// TwinCAT 3 PLC project Library
// Title: lcls-twincat-motion
// Company: SLAC
// ProjectVersion: 0.0.0
// ProgramVersion: 3.1.4026.17
// libraries:
//   LCLS General, * (SLAC)
//   lcls-twincat-math, * (SLAC - LCLS)
//   PMPS, * (SLAC - LCLS)
//   Tc2_EtherCAT, * (Beckhoff Automation GmbH)
//   Tc2_Math, * (Beckhoff Automation GmbH)
//   Tc2_MC2, * (Beckhoff Automation GmbH)
//   Tc2_Standard, * (Beckhoff Automation GmbH)
//   Tc2_System, * (Beckhoff Automation GmbH)
//   Tc2_Utilities, * (Beckhoff Automation GmbH)
//   Tc3_IPCDiag, * (Beckhoff Automation GmbH)
//   Tc3_JsonXml, * (Beckhoff Automation GmbH)
//   Tc3_Module, * (Beckhoff Automation GmbH)
//   TcUnit, * (www.tcunit.org)
// project tree:
//   DUTs/Deprecated/ ENUM_MotionRequest.TcDUT (not stored), DUT_MotionPneumaticActuator.TcDUT (not stored), DUT_MotionStage.TcDUT (not stored), DUT_PositionState.TcDUT (not stored), EL5042_Status.TcDUT (not stored), ENUM_EpicsHomeCmd.TcDUT (not stored), ENUM_EpicsInOut.TcDUT (not stored), ENUM_EpicsInOut_INT.TcDUT (not stored), ENUM_EpicsMotorCmd.TcDUT (not stored), ENUM_MotionFFType.TcDUT (not stored), ENUM_PnuematicActuatorPositionState.TcDUT (not stored), ENUM_StageBrakeMode.TcDUT (not stored), ENUM_StageEnableMode.TcDUT (not stored), ENUM_StatePMPSStatus.TcDUT (not stored)
//   DUTs/DS402/ ENUM_AxisStates.TcDUT (not stored), E_DS402DriveState.TcDUT, E_DS402EGU.TcDUT, E_DS402HomingMethod.TcDUT (not stored), E_DS402OpMode.TcDUT, E_HomeStates.TcDUT (not stored), E_Module.TcDUT (not stored), E_MoveMode.TcDUT (not stored), E_MoveState.TcDUT (not stored), ST_DS402Drive.TcDUT, ST_DS402DriveStatus.TcDUT
//   DUTs/ E_EpicsHomeCmd.TcDUT, ST_AxisParameterSetExposed.TcDUT (not stored), E_LCLSMotionError.TcDUT (not stored), E_MotionFFType.TcDUT (not stored), E_StatePMPSStatus.TcDUT (not stored), ST_MotionEpicsInterface.TcDUT, ST_MotionStage.TcDUT, ST_PositionState.TcDUT, ST_StateEpicsToPlc.TcDUT (not stored), ST_StatePlcToEpics.TcDUT (not stored), ST_StatePMPSEpicsToPlc.TcDUT (not stored), ST_EL5042_Status.TcDUT (not stored), E_EpicsInOut.TcDUT (not stored), E_EpicsMotorCmd.TcDUT, E_MotionRequest.TcDUT (not stored), E_StageBrakeMode.TcDUT (not stored), E_StageEnableMode.TcDUT (not stored), ST_MotionPneumaticActuator.TcDUT (not stored), E_PnuematicActuatorPositionState.TcDUT (not stored), ST_RenishawAbsEnc.TcDUT (not stored), ST_StatePMPSPlcToEpics.TcDUT (not stored)
//   GVLs/ MOTION_GVL.TcGVL (not stored), MotionConstants.TcGVL (not stored)
//   / PlcTask.TcTTO (not stored)
//   POUs/Deprecated/ FB_EpicsInOut.TcPOU (not stored), FB_PositionStateBase.TcPOU (not stored), FB_PositionStateBase_WithPMPS.TcPOU (not stored), FB_PositionStateBase_WithPMPS_Test.TcPOU (not stored), FB_PositionStateInOut.TcPOU (not stored), FB_PositionStateInOut_WithPMPS.TcPOU (not stored), FB_PositionStateInOut_WithPMPS_Test.TcPOU (not stored), FB_PositionStateManager.TcPOU (not stored), FB_PositionStatePMPS.TcPOU (not stored), FB_PositionStatePMPS_Base.TcPOU (not stored), FB_PositionStatePMPS_Test.TcPOU (not stored), FB_StatePTPMove.TcPOU (not stored)
//   POUs/ImplicitChecks/ CheckBounds.TcPOU (not stored), CheckDivDInt.TcPOU (not stored), CheckDivLInt.TcPOU (not stored), CheckDivLReal.TcPOU (not stored), CheckDivReal.TcPOU (not stored)
//   POUs/Motion/DS402/ FB_MotionStageE727.TcPOU, FB_MotionStageMCS2.TcPOU, I_DS402GenericDrive.TcIO
//   POUs/Motion/ FB_EncoderValue.TcPOU (not stored), FB_EncSaveRestore.TcPOU (not stored), FB_LogMotionError.TcPOU (not stored), FB_MotionBacklashCompensation.TcPOU (not stored), FB_MotionHoming.TcPOU (not stored), FB_MotionRequest.TcPOU (not stored), FB_MotionStage.TcPOU, FB_MotionStageNCParams.TcPOU (not stored), FB_MotionStageSim.TcPOU (not stored), FB_MotionPneumaticActuator.TcPOU (not stored), FB_MotionVirtualFrame.TcPOU (not stored)
//   POUs/Motion/Gantry/ FB_GantryAutoCoupling.TcPOU (not stored), FB_GantryDiffVirtualLimitSwitch.TcPOU (not stored)
//   POUs/Motion/PMPS/ FB_EncErrorFFO.TcPOU (not stored), FB_MiscStatesErrorFFO.TcPOU (not stored), FB_MotionBPTM.TcPOU (not stored), FB_MotionClearAsserts.TcPOU (not stored), FB_MotionReadPMPSDBND.TcPOU (not stored), FB_PerMotorFFOND.TcPOU (not stored), FB_NCErrorFFO.TcPOU (not stored), FB_PositionStatePMPS1D.TcPOU (not stored), FB_PositionStatePMPS2D.TcPOU (not stored), FB_PositionStatePMPS3D.TcPOU (not stored), FB_PositionStatePMPSND_Core.TcPOU (not stored), FB_Standard_PMPSDB.TcPOU (not stored), FB_StatePMPSEnables.TcPOU (not stored), FB_StatePMPSEnablesND.TcPOU (not stored)
//   POUs/Motion/States/Examples/ FB_PositionState1D_InOut.TcPOU (not stored), FB_PositionStatePMPS2D_InOut.TcPOU (not stored), FB_PositionStatePMPS1D_InOut.TcPOU (not stored), FB_PositionState2D_InOut.TcPOU (not stored)
//   POUs/Motion/States/ FB_PositionState2D.TcPOU (not stored), FB_PositionState3D.TcPOU (not stored), FB_PositionStateND_Core.TcPOU (not stored), FB_PositionStateMove.TcPOU (not stored), FB_PositionState1D.TcPOU (not stored), FB_PositionStateMoveND.TcPOU (not stored), FB_PositionStateRead.TcPOU (not stored), FB_PositionStateReadND.TcPOU (not stored), FB_StateSetupHelper.TcPOU (not stored), FB_StatesInputHandler.TcPOU (not stored)
//   POUs/Motion/States/Helpers/ FB_RawCountConverter.TcPOU (not stored), F_AtPositionState.TcPOU (not stored), F_PosOverLowerBound.TcPOU (not stored), F_PosUnderUpperBound.TcPOU (not stored), F_PosWithinDelta.TcPOU (not stored)
//   POUs/Motion/States/Internals/ FB_PositionStateInternal.TcPOU (not stored), FB_PositionStateInternalND.TcPOU (not stored), FB_PositionStateLock.TcPOU (not stored)
//   POUs/Motion/Utils/ FB_SetEnables.TcPOU (not stored), F_MotionErrorCodeLookup.TcPOU (not stored)
//   POUs/MotorTesting/ FB_MicroStepCountTest.TcPOU (not stored)
//   tc_mca_std_lib/DUTs/ DUT_AxisStatus_v0_01.TcDUT (not stored)
//   tc_mca_std_lib/GVLs/ GVL.TcGVL (not stored)
//   tc_mca_std_lib/POUs/ChangeConfig/ FB_ReadFloatParameter.TcPOU (not stored), FB_ReadParameterInNc_v1_00.TcPOU (not stored), FB_WriteFloatParameter.TcPOU (not stored), FB_WriteParameterInNc_v1_00.TcPOU (not stored)
//   tc_mca_std_lib/POUs/ErrorHandling/ DUT_ErrorState.TcDUT (not stored), DUT_TerminalError.TcDUT (not stored), FB_ErrorList.TcPOU (not stored), FB_TerminalError.TcPOU (not stored), GVL_ErrorSystem.TcGVL (not stored), ST_ErrorSystem.TcDUT (not stored)
//   tc_mca_std_lib/POUs/Hardware/EtherCAT_Terminals/Analog_Inputs/ EL3174_0002.TcPOU (not stored), EL3214.TcPOU (not stored), EL3255.TcPOU (not stored), FB_CalculateFrequency_3702_v0_01.TcPOU (not stored)
//   tc_mca_std_lib/POUs/Hardware/EtherCAT_Terminals/Digital_Inputs/ EL1008.TcPOU (not stored), EL1018.TcPOU (not stored), EL1808.TcPOU (not stored), EL1809.TcPOU (not stored), EL1819.TcPOU (not stored), FB_EL1252ASM_v1_00.TcPOU (not stored)
//   tc_mca_std_lib/POUs/Hardware/EtherCAT_Terminals/Digital_Outputs/ EL2014.TcPOU (not stored), EL2252.TcPOU (not stored), EL2808.TcPOU (not stored), EL2819.TcPOU (not stored)
//   tc_mca_std_lib/POUs/Hardware/EtherCAT_Terminals/Digital_Outputs/External_Types/ dutEL2521_Ctrl.TcDUT (not stored), dutEL2521_Status.TcDUT (not stored)
//   tc_mca_std_lib/POUs/Hardware/EtherCAT_Terminals/Measuring_Terminals/ EL5002.TcPOU (not stored), EL5021.TcPOU (not stored), EL5042.TcPOU (not stored), EL5101.TcPOU (not stored)
//   tc_mca_std_lib/POUs/Hardware/EtherCAT_Terminals/Motion/ EL7211_v1_00.TcPOU (not stored), EL9576_v1_00.TcPOU (not stored)
//   tc_mca_std_lib/POUs/Hardware/EtherCAT_Terminals/System/ EL9410.TcPOU (not stored), EL9505.TcPOU (not stored)
//   tc_mca_std_lib/POUs/Hardware/Other/ EK1200.TcPOU (not stored)
//   tc_mca_std_lib/POUs/Motion/ FB_DriveVirtual.TcPOU (not stored), FB_NcAxis.TcPOU (not stored)
//   tc_mca_std_lib/POUs/Motion/Homing/ FB_HomeDirect.TcPOU (not stored), FB_HomeFinish.TcPOU (not stored), FB_HomePrepare.TcPOU (not stored), FB_HomeReadNcVelocities.TcPOU (not stored), FB_HomeReadSoftLimEnable.TcPOU (not stored), FB_HomeToSwitch.TcPOU (not stored), FB_HomeVirtual.TcPOU (not stored), FB_HomeWriteNcVelocities.TcPOU (not stored), FB_HomeWriteSoftLimEnable.TcPOU (not stored)
//   Tests/ FB_AtPositionState_Test.TcPOU (not stored), FB_AxisParameterSetExposed_Test.TcPOU (not stored), FB_MiscStatesErrorFFO_Test.TcPOU (not stored), FB_MotionBPTM_Test.TcPOU (not stored), FB_MotionClearAsserts_Test.TcPOU (not stored), FB_MotionReadPMPSDBND_Test.TcPOU (not stored), FB_MotionVirtualFrame_Test.TcPOU (not stored), FB_NCErrorFFO_Test.TcPOU (not stored), FB_PerMotorFFOND_Test.TcPOU (not stored), FB_PositionStateMoveND_Test.TcPOU (not stored), FB_PositionStateMove_Test.TcPOU (not stored), FB_PositionStatePMPSND_Test.TcPOU (not stored), FB_PositionStateReadND_Test.TcPOU (not stored), FB_PositionStateRead_Test.TcPOU (not stored), FB_PositionStateND_Test.TcPOU (not stored), FB_PowerEnableMode_Test.TcPOU (not stored), FB_MotionBacklashCompensation_Test.TcPOU (not stored), FB_StatePMPSEnablesND_Test.TcPOU (not stored), FB_StatePMPSEnables_Test.TcPOU (not stored), FB_StateSetupHelper_Test.TcPOU (not stored), FB_TestHelperSetAndMove_Test.TcPOU (not stored), FB_TestStateInitTiming.TcPOU (not stored), PRG_TEST.TcPOU
//   Tests/Helpers/ E_TestStates.TcDUT (not stored), FB_CauseNCError.TcPOU (not stored), FB_MotionStageSetAndMoveHelper.TcPOU (not stored), FB_MotionStageSetHelper.TcPOU (not stored), FB_MotorTestSuite.TcPOU (not stored), FB_PMPSJsonTestHelper.TcPOU (not stored), FB_TestHelperSetAndMove.TcPOU (not stored)
// real-time tasks:
//   TASK PlcTask: cycle T#10ms, priority 20, ADS port 350
// motion (NC):
//   TASK NC-Task 1 SAF: cycle T#1ms, priority 4, ADS port 501
//   TASK NC-Task 1 SVB: cycle T#10ms, priority 8, ADS port 511
//   AXIS Axis_PositionStateRead_Test (id 3)
//   AXIS Axis_AtPositionState_Test (id 4)
//   AXIS Axis_TestHelperSetAndMove_Test (id 5)
//   AXIS Axis_PositionStateReadND_Test_1 (id 6)
//   AXIS Axis_PositionStateReadND_Test_2 (id 7)
//   AXIS Axis_PositionStateReadND_Test_3 (id 8)
//   AXIS Axis_PositionStateMove_Test (id 9)
//   AXIS Axis_PositionStateMoveND_Test_1 (id 10)
//   AXIS Axis_PositionStateMoveND_Test_2 (id 11)
//   AXIS Axis_PositionStateMoveND_Test_3 (id 12)
//   AXIS Axis_PositionStateND_Test_1 (id 13)
//   AXIS Axis_PositionStateND_Test_2 (id 14)
//   AXIS Axis_PositionStateND_Test_3 (id 15)
//   AXIS Axis_NCErrorFFO_Test (id 16)
//   AXIS Axis_PositionStatePMPSND_Test_1 (id 17)
//   AXIS Axis_PositionStatePMPSND_Test_2 (id 18)
//   AXIS Axis_PositionStatePMPSND_Test_3 (id 19)
//   AXIS Axis_StatePMPSEnable_Test (id 20)
//   AXIS Axis_PositionStateReadND_Test_4 (id 21)
//   AXIS Axis_PositionStateReadND_Test_5 (id 22)
//   AXIS Axis_TestStateInitTiming (id 1)
//   AXIS Axis_AxisParameter_Test (id 2)
//   AXIS Axis_PowerEnableMode_Test (id 29)
//   AXIS Axis_BacklashCompensation_Test (id 30)
//     OtherSettings: AllowMotionCmdToSlave=true
//     encoder EncType=1
//       ActPosCorrection: Enable=true
//     drive DrvType=5
//       Analog: TorqueSetpointScale=10, ScaleFactorActTorque=0.1
//       TimeComp: TaskDelayCycles=1
//     controller CtrType=1
//       CtrPara: PriorControlFactor=1
//         Observer: BandWidth=20
//   AXIS Axis_HomeNC_Test1 (id 32)
//     OtherSettings: AllowMotionCmdToSlave=true
//     encoder EncType=1
//     drive DrvType=5
//       Analog: TorqueSetpointScale=10, ScaleFactorActTorque=0.1
//       TimeComp: TaskDelayCycles=1
//     controller CtrType=1
//       CtrPara: PriorControlFactor=1
//         Observer: BandWidth=20
//   AXIS Axis_HomeNC_Test2 (id 33)
//     OtherSettings: AllowMotionCmdToSlave=true
//     encoder EncType=1
//     drive DrvType=5
//       Analog: TorqueSetpointScale=10, ScaleFactorActTorque=0.1
//       TimeComp: TaskDelayCycles=1
//     controller CtrType=1
//       CtrPara: PriorControlFactor=1
//         Observer: BandWidth=20
//   AXIS Axis_HomeNC_Test3 (id 34)
//     OtherSettings: AllowMotionCmdToSlave=true
//     encoder EncType=1
//     drive DrvType=5
//       Analog: TorqueSetpointScale=10, ScaleFactorActTorque=0.1
//       TimeComp: TaskDelayCycles=1
//     controller CtrType=1
//       CtrPara: PriorControlFactor=1
//         Observer: BandWidth=20
//   AXIS Axis_HomeNC_Test4 (id 35)
//     OtherSettings: AllowMotionCmdToSlave=true
//     encoder EncType=1
//     drive DrvType=5
//       Analog: TorqueSetpointScale=10, ScaleFactorActTorque=0.1
//       TimeComp: TaskDelayCycles=1
//     controller CtrType=1
//       CtrPara: PriorControlFactor=1
//         Observer: BandWidth=20
//   AXIS Axis_HomeNC_Test5 (id 36)
//     OtherSettings: AllowMotionCmdToSlave=true
//     encoder EncType=1
//     drive DrvType=5
//       Analog: TorqueSetpointScale=10, ScaleFactorActTorque=0.1
//       TimeComp: TaskDelayCycles=1
//     controller CtrType=1
//       CtrPara: PriorControlFactor=1
//         Observer: BandWidth=20
//   AXIS Axis_HomeNC_Test6 (id 37)
//     OtherSettings: AllowMotionCmdToSlave=true
//     encoder EncType=1
//     drive DrvType=5
//       Analog: TorqueSetpointScale=10, ScaleFactorActTorque=0.1
//       TimeComp: TaskDelayCycles=1
//     controller CtrType=1
//       CtrPara: PriorControlFactor=1
//         Observer: BandWidth=20
//   AXIS Axis_HomeNC_Test7 (id 38)
//     OtherSettings: AllowMotionCmdToSlave=true
//     encoder EncType=1
//     drive DrvType=5
//       Analog: TorqueSetpointScale=10, ScaleFactorActTorque=0.1
//       TimeComp: TaskDelayCycles=1
//     controller CtrType=1
//       CtrPara: PriorControlFactor=1
//         Observer: BandWidth=20
//   AXIS Axis_HomeNC_Test8 (id 39)
//     OtherSettings: AllowMotionCmdToSlave=true
//     encoder EncType=1
//     drive DrvType=5
//       Analog: TorqueSetpointScale=10, ScaleFactorActTorque=0.1
//       TimeComp: TaskDelayCycles=1
//     controller CtrType=1
//       CtrPara: PriorControlFactor=1
//         Observer: BandWidth=20
//   AXIS Axis_McMotionBlocks_Test1 (id 40)
//     OtherSettings: AllowMotionCmdToSlave=true
//     encoder EncType=1
//     drive DrvType=5
//       Analog: TorqueSetpointScale=10, ScaleFactorActTorque=0.1
//       TimeComp: TaskDelayCycles=1
//     controller CtrType=1
//       CtrPara: PriorControlFactor=1
//         Observer: BandWidth=20
//   AXIS Axis_McMotionBlocks_Test2 (id 41)
//     OtherSettings: AllowMotionCmdToSlave=true
//     encoder EncType=1
//     drive DrvType=5
//       Analog: TorqueSetpointScale=10, ScaleFactorActTorque=0.1
//       TimeComp: TaskDelayCycles=1
//     controller CtrType=1
//       CtrPara: PriorControlFactor=1
//         Observer: BandWidth=20
//   AXIS Axis_McMotionBlocks_Test3 (id 42)
//     OtherSettings: AllowMotionCmdToSlave=true
//     encoder EncType=1
//     drive DrvType=5
//       Analog: TorqueSetpointScale=10, ScaleFactorActTorque=0.1
//       TimeComp: TaskDelayCycles=1
//     controller CtrType=1
//       CtrPara: PriorControlFactor=1
//         Observer: BandWidth=20
//   AXIS Axis_McMotionBlocks_Test4 (id 43)
//     OtherSettings: AllowMotionCmdToSlave=true
//     encoder EncType=1
//     drive DrvType=5
//       Analog: TorqueSetpointScale=10, ScaleFactorActTorque=0.1
//       TimeComp: TaskDelayCycles=1
//     controller CtrType=1
//       CtrPara: PriorControlFactor=1
//         Observer: BandWidth=20
//   AXIS Axis_McMotionBlocks_Test5 (id 44)
//     OtherSettings: AllowMotionCmdToSlave=true
//     encoder EncType=1
//     drive DrvType=5
//       Analog: TorqueSetpointScale=10, ScaleFactorActTorque=0.1
//       TimeComp: TaskDelayCycles=1
//     controller CtrType=1
//       CtrPara: PriorControlFactor=1
//         Observer: BandWidth=20
//   AXIS Axis_McMotionBlocks_Test6 (id 45)
//     OtherSettings: AllowMotionCmdToSlave=true
//     encoder EncType=1
//       ActPosCorrection: Enable=true
//     drive DrvType=5
//       Analog: TorqueSetpointScale=10, ScaleFactorActTorque=0.1
//       TimeComp: TaskDelayCycles=1
//     controller CtrType=1
//       CtrPara: PriorControlFactor=1
//         Observer: BandWidth=20
//   AXIS Axis_McMotionBlocks_Test7 (id 46)
//     OtherSettings: AllowMotionCmdToSlave=true
//     encoder EncType=1
//       ActPosCorrection: Enable=true
//     drive DrvType=5
//       Analog: TorqueSetpointScale=10, ScaleFactorActTorque=0.1
//       TimeComp: TaskDelayCycles=1
//     controller CtrType=1
//       CtrPara: PriorControlFactor=1
//         Observer: BandWidth=20
//   AXIS Axis_McMotionBlocks_Test8 (id 47)
//     OtherSettings: AllowMotionCmdToSlave=true
//     encoder EncType=1
//       ActPosCorrection: Enable=true
//     drive DrvType=5
//       Analog: TorqueSetpointScale=10, ScaleFactorActTorque=0.1
//       TimeComp: TaskDelayCycles=1
//     controller CtrType=1
//       CtrPara: PriorControlFactor=1
//         Observer: BandWidth=20
//   AXIS Axis_MotionVirtualFrameRx_Test (id 23)
//   AXIS Axis_MotionVirtualFrameRy_Test (id 24)
//   AXIS Axis_MotionVirtualFrameRz_Test (id 25)
//   AXIS Axis_MotionVirtualFrameVx_Test (id 26)
//   AXIS Axis_MotionVirtualFrameVy_Test (id 27)
//   AXIS Axis_MotionVirtualFrameVz_Test (id 28)
// variable links:
//   Library Instance <-> NC-Task 1 SAF/Axes/Axis_AtPositionState_Test
//     PlcTask Inputs/PRG_TEST.fb_AtPositionState_Test.stMotionStage.Axis.NcToPlc <-> Outputs/ToPlc
//     PlcTask Outputs/PRG_TEST.fb_AtPositionState_Test.stMotionStage.Axis.PlcToNc <-> Inputs/FromPlc
//   Library Instance <-> NC-Task 1 SAF/Axes/Axis_AxisParameter_Test
//     PlcTask Inputs/PRG_TEST.fb_AxisParameterSetExposed_Test.stMotionStage.Axis.NcToPlc <-> Outputs/ToPlc
//     PlcTask Outputs/PRG_TEST.fb_AxisParameterSetExposed_Test.stMotionStage.Axis.PlcToNc <-> Inputs/FromPlc
//   Library Instance <-> NC-Task 1 SAF/Axes/Axis_BacklashCompensation_Test
//     PlcTask Inputs/PRG_TEST.fb_MotionBacklashCompensation_Test.stMotionStage.Axis.NcToPlc <-> Outputs/ToPlc
//     PlcTask Outputs/PRG_TEST.fb_MotionBacklashCompensation_Test.stMotionStage.Axis.PlcToNc <-> Inputs/FromPlc
//   Library Instance <-> NC-Task 1 SAF/Axes/Axis_MotionVirtualFrameRx_Test
//     PlcTask Inputs/PRG_TEST.fbMotionVirtualFrameTest.stMotionStageRx.Axis.NcToPlc <-> Outputs/ToPlc
//     PlcTask Outputs/PRG_TEST.fbMotionVirtualFrameTest.stMotionStageRx.Axis.PlcToNc <-> Inputs/FromPlc
//   Library Instance <-> NC-Task 1 SAF/Axes/Axis_MotionVirtualFrameRy_Test
//     PlcTask Inputs/PRG_TEST.fbMotionVirtualFrameTest.stMotionStageRy.Axis.NcToPlc <-> Outputs/ToPlc
//     PlcTask Outputs/PRG_TEST.fbMotionVirtualFrameTest.stMotionStageRy.Axis.PlcToNc <-> Inputs/FromPlc
//   Library Instance <-> NC-Task 1 SAF/Axes/Axis_MotionVirtualFrameRz_Test
//     PlcTask Inputs/PRG_TEST.fbMotionVirtualFrameTest.stMotionStageRz.Axis.NcToPlc <-> Outputs/ToPlc
//     PlcTask Outputs/PRG_TEST.fbMotionVirtualFrameTest.stMotionStageRz.Axis.PlcToNc <-> Inputs/FromPlc
//   Library Instance <-> NC-Task 1 SAF/Axes/Axis_MotionVirtualFrameVx_Test
//     PlcTask Inputs/PRG_TEST.fbMotionVirtualFrameTest.stMotionStageVx.Axis.NcToPlc <-> Outputs/ToPlc
//     PlcTask Outputs/PRG_TEST.fbMotionVirtualFrameTest.nPositionCountsVx <-> Enc/Inputs/In/nDataIn1
//     PlcTask Outputs/PRG_TEST.fbMotionVirtualFrameTest.stMotionStageVx.Axis.PlcToNc <-> Inputs/FromPlc
//   Library Instance <-> NC-Task 1 SAF/Axes/Axis_MotionVirtualFrameVy_Test
//     PlcTask Inputs/PRG_TEST.fbMotionVirtualFrameTest.stMotionStageVy.Axis.NcToPlc <-> Outputs/ToPlc
//     PlcTask Outputs/PRG_TEST.fbMotionVirtualFrameTest.nPositionCountsVy <-> Enc/Inputs/In/nDataIn1
//     PlcTask Outputs/PRG_TEST.fbMotionVirtualFrameTest.stMotionStageVy.Axis.PlcToNc <-> Inputs/FromPlc
//   Library Instance <-> NC-Task 1 SAF/Axes/Axis_MotionVirtualFrameVz_Test
//     PlcTask Inputs/PRG_TEST.fbMotionVirtualFrameTest.stMotionStageVz.Axis.NcToPlc <-> Outputs/ToPlc
//     PlcTask Outputs/PRG_TEST.fbMotionVirtualFrameTest.nPositionCountsVz <-> Enc/Inputs/In/nDataIn1
//     PlcTask Outputs/PRG_TEST.fbMotionVirtualFrameTest.stMotionStageVz.Axis.PlcToNc <-> Inputs/FromPlc
//   Library Instance <-> NC-Task 1 SAF/Axes/Axis_NCErrorFFO_Test
//     PlcTask Inputs/PRG_TEST.fb_NCErrorFFO_Test.stMotionStage.Axis.NcToPlc <-> Outputs/ToPlc
//     PlcTask Outputs/PRG_TEST.fb_NCErrorFFO_Test.stMotionStage.Axis.PlcToNc <-> Inputs/FromPlc
//   Library Instance <-> NC-Task 1 SAF/Axes/Axis_PositionStateMoveND_Test_1
//     PlcTask Inputs/PRG_TEST.fb_PositionStateMoveND_Test.astMotionStage[1].Axis.NcToPlc <-> Outputs/ToPlc
//     PlcTask Outputs/PRG_TEST.fb_PositionStateMoveND_Test.astMotionStage[1].Axis.PlcToNc <-> Inputs/FromPlc
//   Library Instance <-> NC-Task 1 SAF/Axes/Axis_PositionStateMoveND_Test_2
//     PlcTask Inputs/PRG_TEST.fb_PositionStateMoveND_Test.astMotionStage[2].Axis.NcToPlc <-> Outputs/ToPlc
//     PlcTask Outputs/PRG_TEST.fb_PositionStateMoveND_Test.astMotionStage[2].Axis.PlcToNc <-> Inputs/FromPlc
//   Library Instance <-> NC-Task 1 SAF/Axes/Axis_PositionStateMoveND_Test_3
//     PlcTask Inputs/PRG_TEST.fb_PositionStateMoveND_Test.astMotionStage[3].Axis.NcToPlc <-> Outputs/ToPlc
//     PlcTask Outputs/PRG_TEST.fb_PositionStateMoveND_Test.astMotionStage[3].Axis.PlcToNc <-> Inputs/FromPlc
//   Library Instance <-> NC-Task 1 SAF/Axes/Axis_PositionStateMove_Test
//     PlcTask Inputs/PRG_TEST.fb_PositionStateMove_Test.stMotionStage.Axis.NcToPlc <-> Outputs/ToPlc
//     PlcTask Outputs/PRG_TEST.fb_PositionStateMove_Test.stMotionStage.Axis.PlcToNc <-> Inputs/FromPlc
//   Library Instance <-> NC-Task 1 SAF/Axes/Axis_PositionStateND_Test_1
//     PlcTask Inputs/PRG_TEST.fb_PositionStateND_Test.stMotionStage1.Axis.NcToPlc <-> Outputs/ToPlc
//     PlcTask Outputs/PRG_TEST.fb_PositionStateND_Test.stMotionStage1.Axis.PlcToNc <-> Inputs/FromPlc
//   Library Instance <-> NC-Task 1 SAF/Axes/Axis_PositionStateND_Test_2
//     PlcTask Inputs/PRG_TEST.fb_PositionStateND_Test.stMotionStage2.Axis.NcToPlc <-> Outputs/ToPlc
//     PlcTask Outputs/PRG_TEST.fb_PositionStateND_Test.stMotionStage2.Axis.PlcToNc <-> Inputs/FromPlc
//   Library Instance <-> NC-Task 1 SAF/Axes/Axis_PositionStateND_Test_3
//     PlcTask Inputs/PRG_TEST.fb_PositionStateND_Test.stMotionStage3.Axis.NcToPlc <-> Outputs/ToPlc
//     PlcTask Outputs/PRG_TEST.fb_PositionStateND_Test.stMotionStage3.Axis.PlcToNc <-> Inputs/FromPlc
//   Library Instance <-> NC-Task 1 SAF/Axes/Axis_PositionStatePMPSND_Test_1
//     PlcTask Inputs/PRG_TEST.fb_PositionStatePMPSND_Test.stMotionStage1.Axis.NcToPlc <-> Outputs/ToPlc
//     PlcTask Outputs/PRG_TEST.fb_PositionStatePMPSND_Test.stMotionStage1.Axis.PlcToNc <-> Inputs/FromPlc
//   Library Instance <-> NC-Task 1 SAF/Axes/Axis_PositionStatePMPSND_Test_2
//     PlcTask Inputs/PRG_TEST.fb_PositionStatePMPSND_Test.stMotionStage2.Axis.NcToPlc <-> Outputs/ToPlc
//     PlcTask Outputs/PRG_TEST.fb_PositionStatePMPSND_Test.stMotionStage2.Axis.PlcToNc <-> Inputs/FromPlc
//   Library Instance <-> NC-Task 1 SAF/Axes/Axis_PositionStatePMPSND_Test_3
//     PlcTask Inputs/PRG_TEST.fb_PositionStatePMPSND_Test.stMotionStage3.Axis.NcToPlc <-> Outputs/ToPlc
//     PlcTask Outputs/PRG_TEST.fb_PositionStatePMPSND_Test.stMotionStage3.Axis.PlcToNc <-> Inputs/FromPlc
//   Library Instance <-> NC-Task 1 SAF/Axes/Axis_PositionStateReadND_Test_1
//     PlcTask Inputs/PRG_TEST.fb_PositionStateReadND_Test.astMotionStage[1].Axis.NcToPlc <-> Outputs/ToPlc
//     PlcTask Outputs/PRG_TEST.fb_PositionStateReadND_Test.astMotionStage[1].Axis.PlcToNc <-> Inputs/FromPlc
//   Library Instance <-> NC-Task 1 SAF/Axes/Axis_PositionStateReadND_Test_2
//     PlcTask Inputs/PRG_TEST.fb_PositionStateReadND_Test.astMotionStage[2].Axis.NcToPlc <-> Outputs/ToPlc
//     PlcTask Outputs/PRG_TEST.fb_PositionStateReadND_Test.astMotionStage[2].Axis.PlcToNc <-> Inputs/FromPlc
//   Library Instance <-> NC-Task 1 SAF/Axes/Axis_PositionStateReadND_Test_3
//     PlcTask Inputs/PRG_TEST.fb_PositionStateReadND_Test.astMotionStage[3].Axis.NcToPlc <-> Outputs/ToPlc
//     PlcTask Outputs/PRG_TEST.fb_PositionStateReadND_Test.astMotionStage[3].Axis.PlcToNc <-> Inputs/FromPlc
//   Library Instance <-> NC-Task 1 SAF/Axes/Axis_PositionStateReadND_Test_4
//     PlcTask Inputs/PRG_TEST.fb_PositionStateReadND_Test.astSqMotionStage[1].Axis.NcToPlc <-> Outputs/ToPlc
//     PlcTask Outputs/PRG_TEST.fb_PositionStateReadND_Test.astSqMotionStage[1].Axis.PlcToNc <-> Inputs/FromPlc
//   Library Instance <-> NC-Task 1 SAF/Axes/Axis_PositionStateReadND_Test_5
//     PlcTask Inputs/PRG_TEST.fb_PositionStateReadND_Test.astSqMotionStage[2].Axis.NcToPlc <-> Outputs/ToPlc
//     PlcTask Outputs/PRG_TEST.fb_PositionStateReadND_Test.astSqMotionStage[2].Axis.PlcToNc <-> Inputs/FromPlc
//   Library Instance <-> NC-Task 1 SAF/Axes/Axis_PositionStateRead_Test
//     PlcTask Inputs/PRG_TEST.fb_PositionStateRead_Test.stMotionStage.Axis.NcToPlc <-> Outputs/ToPlc
//     PlcTask Outputs/PRG_TEST.fb_PositionStateRead_Test.stMotionStage.Axis.PlcToNc <-> Inputs/FromPlc
//   Library Instance <-> NC-Task 1 SAF/Axes/Axis_PowerEnableMode_Test
//     PlcTask Inputs/PRG_TEST.fb_PowerEnableMode_Test.stMotionStage.Axis.NcToPlc <-> Outputs/ToPlc
//     PlcTask Outputs/PRG_TEST.fb_PowerEnableMode_Test.stMotionStage.Axis.PlcToNc <-> Inputs/FromPlc
//   Library Instance <-> NC-Task 1 SAF/Axes/Axis_StatePMPSEnable_Test
//     PlcTask Inputs/PRG_TEST.fb_StatePMPSEnables_Test.stMotionStage.Axis.NcToPlc <-> Outputs/ToPlc
//     PlcTask Outputs/PRG_TEST.fb_StatePMPSEnables_Test.stMotionStage.Axis.PlcToNc <-> Inputs/FromPlc
//   Library Instance <-> NC-Task 1 SAF/Axes/Axis_TestHelperSetAndMove_Test
//     PlcTask Inputs/PRG_TEST.fb_TestHelperSetAndMove_Test.stMotionStage.Axis.NcToPlc <-> Outputs/ToPlc
//     PlcTask Outputs/PRG_TEST.fb_TestHelperSetAndMove_Test.stMotionStage.Axis.PlcToNc <-> Inputs/FromPlc
//   Library Instance <-> NC-Task 1 SAF/Axes/Axis_TestStateInitTiming
//     PlcTask Inputs/PRG_TEST.fb_TestStateInitTiming.stMotionStage.Axis.NcToPlc <-> Outputs/ToPlc
//     PlcTask Outputs/PRG_TEST.fb_TestStateInitTiming.stMotionStage.Axis.PlcToNc <-> Inputs/FromPlc

// ---- DUTs/DS402/E_DS402DriveState.TcDUT
{attribute 'qualified_only'}
{attribute 'strict'}
{attribute 'to_string'}
TYPE E_DS402DriveState :
(
    INIT:=0,
    NO_FAULT:=1,
    SWITCH_ON_READY:=2,
    SWITCH_ON:=3,
    OPERATION_ENABLED:=4,
    FAULT:=5,
    FAULT_ACTIVE:=6,
    QUICK_STOP_ACTIVE:=7,
    SWITCH_ON_DISABLED:=8,
    MODE_ERROR:=9,
    WAIT	:= 10,
    DONE:=11
) UINT;
END_TYPE

// ---- DUTs/DS402/E_DS402EGU.TcDUT
{attribute 'qualified_only'}
{attribute 'strict'}
{attribute 'to_string'}
TYPE E_DS402EGU :
(
    MM:=0,
    UM:=1,
    NM:=2
);
END_TYPE

// ---- DUTs/DS402/E_DS402OpMode.TcDUT
{attribute 'qualified_only'}
{attribute 'strict'}
{attribute 'to_string'}
TYPE E_DS402OpMode :
(
    NONE:= 0,
    CALIBRATION:=-1,
    MCS2_OL_SM:=-4,
    PROFILE_POSITION:=1,
    HOMING:=6,
    CSP:=8
) SINT;
END_TYPE

// ---- DUTs/DS402/ST_DS402Drive.TcDUT
TYPE ST_DS402Drive:
STRUCT
    (* Global variables for the TPDO data from the drive. Each one is linked to the respective TPDO channel. *)
    stDS402DriveStatus 		AT %I*	: 	ST_DS402DriveStatus;
    nModeOfOperationDisplay AT %I*	: 	SINT;
    //nActualPosition 		AT %I*	: 	DINT;
    (*CSP drive mode*)
    nFollowingError 		AT %I*	: 	DINT;
    (* Global variables for the RPDO data to the drive. Each one is linked to the respective RPDO channel. *)
    // connected to I/O Task 'Control Word'
    nDS402DriveControl		AT %Q*	:	UINT;
    // Connected to NC task Ctrl 1 and Ctrl 2
    nDS402DriveControlNC	AT %I*	:	UINT;
    nTargetPosition 		AT %Q* 	: 	DINT;
    nModeOfOperation 		AT %Q* 	: 	SINT;
    nModeOfOperationNC 		AT %I* 	: 	SINT;
    (* Global variables for the RPDO data to the drive. Each one is linked to the respective RPDO channel. *)
    nProfilVelocity 		AT %Q* 	: 	DINT;
    nProfilAcceleration		AT %Q* 	: 	DINT;
    nProfilDecceleration	AT %Q* 	: 	DINT;
    nVelocityActualValue	AT %Q* 	: 	DINT;
    (* Global variables for the TPDO data from the drive. Each one is linked to the respective TPDO channel. *)
    nScantargetPosition		AT %Q*	: 	DINT;
    uScantargetVelocity		AT %Q*	: 	ULINT;
    (* Port Number of EtherCAT Slave *)
    nSlaveAddr	AT %I*  : UINT;
END_STRUCT
END_TYPE

// ---- DUTs/DS402/ST_DS402DriveStatus.TcDUT
TYPE ST_DS402DriveStatus :
    STRUCT
        ReadyToSwitchOn			: BIT; (* Bit 0 *)
        SwitchedOn				: BIT; (* Bit 1 *)
        OperationEnabled		: BIT; (* Bit 2 *)
        Fault					: BIT; (* Bit 3 *)
        VoltageEnabled			: BIT; (* Bit 4 *)
        QuickStopActive			: BIT; (* Bit 5 *)
        SwitchOnDisabled		: BIT; (* Bit 6 *)
        WarningCondition		: BIT; (* Bit 7 *)
        TrajectoryAborted		: BIT; (* Bit 8 *)
        RemoteCANopenControl	: BIT; (* Bit 9 *)
        TargetReached			: BIT; (* Bit 10 *)
        InternalLimitActive		: BIT; (* Bit 11 *)
        Bit12_OpModeSpecific	: BIT; (* Bit 12 *)
        Bit13_OpModeSpecific	: BIT; (* Bit 13 *)

    END_STRUCT
END_TYPE

// ---- DUTs/E_EpicsHomeCmd.TcDUT
{attribute 'qualified_only'}
{attribute 'strict'}
TYPE E_EpicsHomeCmd :
    // Defines the valid options for homing in FB_MotionStage
(
    LOW_LIMIT:=1, // Low limit switch
    HIGH_LIMIT:=2, // High limit switch
    HOME_VIA_LOW:=3, // Home switch via low switch
    HOME_VIA_HIGH:=4, // Home switch via high switch
    AUTO_ZERO	:= 5,	// Piezo Drives Homing
    ABSOLUTE_SET:=15, // Set here to be fHomePosition
    NONE:=-1 // Do not home, ever
);
END_TYPE

// ---- DUTs/ST_MotionEpicsInterface.TcDUT
TYPE ST_MotionEpicsInterface :
    // Defines the EPICS interface to moving a motor in TwinCAT
STRUCT
    // Name to use for log messages, fast faults, etc.
    sName: STRING;
    // Set to gantry difference tolerance
    nGantryTol: LINT:=0;
    // Encoder count at which this axis is aligned with other axis
    nEncRef: ULINT:=0;

    (* Commands *)
    // Used internally to request enables
    bEnable: BOOL;

    // Used internally to reset errors and other state
    {attribute 'pytmc' := '
        pv: PLC:bReset
        io: io
        field: ZNAM FALSE
        field: ONAM TRUE
        field: DESC Used internally to reset errors
    '}
    bReset: BOOL;
    // Used internally and by the IOC to start or stop a move
    bExecute: BOOL;

    (* Command Args *)
    // Used internally and by the IOC to pick what kind of move to do
    nCommand: INT;
    // Used internally and by the IOC to pass additional data to some commands
    nCmdData: INT;
    // Used internally and by the IOC to pick a destination for the move
    fPosition: LREAL;
    // Used internally and by the IOC to pick a move velocity
    fVelocity: LREAL;
    // Used internally and by the IOC to pick a move acceleration
    fAcceleration: LREAL;
    // Used internally and by the IOC to pick a move deceleration
    fDeceleration: LREAL;
    // Used internally and by the IOC to pick a home position
    {attribute 'pytmc' := '
        pv: PLC:fHomePosition
        io: io
        field: DESC Used internally and by the IOC to pick home position
    '}
    fHomePosition: LREAL;

    (* Info *)
    // Unique ID assigned to each axis in the NC
    nMotionAxisID: UDINT:=0;
    (* Returns *)
    // TRUE if in the middle of a command
    bBusy: BOOL;
    // TRUE if we've done a command and it has finished
    bDone: BOOL;
    // TRUE if the motor has been homed, or does not need to be homed
    bHomed: BOOL;

    // TRUE if we're in an error state
    {attribute 'pytmc' := '
        pv: PLC:bError
        io: i
        field: ZNAM FALSE
        field: ONAM TRUE
        field: DESC TRUE if we are in an error state
        update: 100Hz notify
    '}
    bError: BOOL;
    // Error code if nonzero
    {attribute 'pytmc' := '
        pv: PLC:nErrorId
        io: i
        field: DESC Error code if nonzero
        update: 100Hz notify
    '}
    nErrorId: UDINT;
    // Message to identify the error state
    {attribute 'pytmc' := '
        pv: PLC:sErrorMessage
        io: i
        field: DESC Message to identify the error state
        update: 100Hz notify
    '}
    sErrorMessage: STRING;

  // Misc axis status information for the IOC
    stAxisStatus: DUT_AxisStatus_v0_01;
END_STRUCT
END_TYPE

// ---- DUTs/ST_MotionStage.TcDUT
TYPE ST_MotionStage :
    // Defines the EPICS interface to moving a motor in TwinCAT
STRUCT
    (* Hardware *)

    // PLC Axis Reference
    Axis: AXIS_REF;
    // NC Forward Limit Switch: TRUE if ok to move
    bLimitForwardEnable AT %I*: BOOL;
    // NC Backward Limit Switch: TRUE if ok to move
    bLimitBackwardEnable AT %I*: BOOL;
    // NO Home Switch: TRUE if at home
    bHome AT %I*: BOOL;
    // NC Brake Output: TRUE to release brake
    bBrakeRelease AT %Q*: BOOL;
    // NC STO Input: TRUE if ok to move
    {attribute 'pytmc' := '
        pv: PLC:bHardwareEnable
        io: i
        field: ZNAM FALSE
        field: ONAM TRUE
        field: DESC TRUE if STO not hit
    '}
    bHardwareEnable AT %I*: BOOL;

    // Raw encoder IO for ULINT (Biss-C)
    nRawEncoderULINT AT %I*: ULINT;
    // Raw encoder IO for UINT (Relative Encoders)
    nRawEncoderUINT AT %I*: UINT;
    // Raw encoder IO for INT (LVDT)
    nRawEncoderINT AT %I*: INT;
    // Raw encoder IO for INT (EL5072 LVDT)
    nRawEncoderDINT AT %I*: DINT;

    (* Psuedo-hardware *)

    // Forward enable EPS summary
    bAllForwardEnable: BOOL:=FALSE;
    // Backward enable EPS summary
    bAllBackwardEnable: BOOL:=FALSE;
    // Enable EPS summary encapsulating emergency stop button and any additional motion preventive hardware
    bAllEnable: BOOL:=FALSE;
    // Forward virtual gantry limit switch
    bGantryForwardEnable: BOOL:=FALSE;
    // Backward virtual gantry limit switch
    bGantryBackwardEnable: BOOL:=FALSE;
    // Encoder count summary, if linked above
    {attribute 'pytmc' := '
        pv: PLC:nEncoderCount
        io: i
        field: DESC Count from encoder hardware
    '}
    nEncoderCount: UDINT;
    // Forward Enable EPS struct
    {attribute 'pytmc' := '
        pv: PLC:stEPSF
        io: i
        field: DESC Forward Enable Interlocks
    '}
    stEPSForwardEnable: DUT_EPS;
    // Backward Enable EPS struct
    {attribute 'pytmc' := '
        pv: PLC:stEPSB
        io: i
        field: DESC Backward Enable Interlocks
    '}
    stEPSBackwardEnable: DUT_EPS;
    // Power Enable EPS struct
    {attribute 'pytmc' := '
        pv: PLC:stEPSP
        io: i
        field: DESC Power Interlocks
    '}
    stEPSPowerEnable: DUT_EPS;

    (* Settings *)
    // Name to use for log messages, fast faults, etc.
    sName: STRING;
    // If TRUE, we want to enable the motor independently of PMPS or other safety systems.
    bPowerSelf: BOOL:=FALSE;
    // Determines when we automatically enable the motor
    nEnableMode: E_StageEnableMode:=E_StageEnableMode.DURING_MOTION;
    // Determines when we automatically disengage the brake
    nBrakeMode: E_StageBrakeMode:=E_StageBrakeMode.IF_ENABLED;
    // Determines our encoder homing strategy
    nHomingMode: E_EpicsHomeCmd:=E_EpicsHomeCmd.NONE;
    // Set true to activate gantry EPS
    bGantryAxis: BOOL:=FALSE;

    // Set to gantry difference tolerance
    nGantryTol: LINT:=0;

    // Encoder count at which this axis is aligned with other axis
    nEncRef: ULINT:=0;

    (* Commands *)
    // Used internally to request enables
    bEnable: BOOL;
    // Used internally to reset errors and other state
    {attribute 'pytmc' := '
        pv: PLC:bReset
        io: io
        field: ZNAM FALSE
        field: ONAM TRUE
        field: DESC Used internally to reset errors
    '}
    bReset: BOOL;
    // Used internally and by the IOC to start or stop a move
    bExecute: BOOL;
    // Used by the IOC to disable an axis
    {attribute 'pytmc' := '
        pv: PLC:bUserEnable
        io: io
        field: ZNAM DISABLE
        field: ONAM ENABLE
        field: DESC Used to disable power entirely for an axis
        autosave_pass1: VAL
    '}
    bUserEnable: BOOL := 1;

    (* Shortcut Commands *)
    // Start a move to fPosition with fVelocity
    bMoveCmd: BOOL;
    // Start the homing routine
    {attribute 'pytmc' := '
        pv: PLC:bHomeCmd
        io: io
        field: DESC Start the homing routine
    '}
    bHomeCmd: BOOL;

    (* Command Args *)
    // Used internally and by the IOC to pick what kind of move to do
    nCommand: INT;
    // Used internally and by the IOC to pass additional data to some commands
    nCmdData: INT;
    // Used internally and by the IOC to pick a destination for the move
    fPosition: LREAL;
    // Used internally and by the IOC to pick a move velocity
    fVelocity: LREAL;
    // Used internally and by the IOC to pick a move acceleration
    fAcceleration: LREAL;
    // Used internally and by the IOC to pick a move deceleration
    fDeceleration: LREAL;
    // Used internally and by the IOC to pick a home position
    {attribute 'pytmc' := '
        pv: PLC:fHomePosition
        io: io
        field: DESC Used internally and by the IOC to pick home position
        autosave_pass1: VAL
    '}
    fHomePosition: LREAL;

    (* Info *)
    // Unique ID assigned to each axis in the NC
    nMotionAxisID: UDINT:=0;

    (* Returns *)
    // TRUE if done enabling
    bEnableDone: BOOL;
    // TRUE if in the middle of a command
    bBusy: BOOL;
    // TRUE if we've done a command and it has finished
    bDone: BOOL;
    // TRUE if the motor has been homed, or does not need to be homed
    bHomed: BOOL;
    // TRUE if we have safety permission to move
    bSafetyReady: BOOL;
    // TRUE if we're in an error state
    {attribute 'pytmc' := '
        pv: PLC:bError
        io: i
        field: ZNAM FALSE
        field: ONAM TRUE
        field: DESC TRUE if we are in an error state
    '}
    bError: BOOL;
    // Error code if nonzero
    {attribute 'pytmc' := '
        pv: PLC:nErrorId
        io: i
        field: DESC Error code if nonzero
    '}
    nErrorId: UDINT;
    // Message to identify the error state
    {attribute 'pytmc' := '
        pv: PLC:sErrorMessage
        io: i
        field: DESC Message to identify the error state
    '}
    sErrorMessage: STRING;
    // Internal hook for custom error messages
    sCustomErrorMessage: STRING;
    // MC_ReadParameterSet Output
    stAxisParameters: ST_AxisParameterSet;
    // NC parameters that are exposed with pytmc pragmas
    {attribute 'pytmc' := '
        pv: PLC:AxisPar
        io: i
        field: DESC Axis configuration parameters in the numerical controller.
    '}
    stAxisParametersExposed: ST_AxisParameterSetExposed;
    // True if we've updated stAxisParameters at least once
    bAxisParamsInit: BOOL;

    // Misc axis status information for the IOC
    stAxisStatus: DUT_AxisStatus_v0_01;

    (* Other status information for users of the IOC *)
    // Position lag difference
    {attribute 'pytmc' := '
        pv: PLC:fPosDiff
        io: i
        field: DESC Position lag difference
    '}
    fPosDiff: LREAL;

    (* Backlash compensation*)
    // Enabled axis backlash compensation
    {attribute 'pytmc' := '
        pv: PLC:bBacklashEn
        io: io
        field: ZNAM FALSE
        field: ONAM TRUE
        field: DESC Enable Backlash compensation
        autosave_pass1: VAL
    '}
    bUserBacklashEn: BOOL;

    // backlash compensation status
    {attribute 'pytmc' := '
        pv: PLC:bBacklasStatus
        io: i
        field: ZNAM DISABLED
        field: ONAM ENABLED
        field: DESC Backlash compensation status
    '}
    bBacklashStatus: BOOL;

    // Backlash compensation value
    {attribute 'pytmc' := '
        pv: PLC:fBacklash
        io: io
        field: DESC Backlash compensation
        autosave_pass1: VAL
    '}
    fBacklash: LREAL;

    // Current Backlash compensation value ?
    {attribute 'pytmc' := '
        pv: PLC:fCurrentBacklash
        io: i
        field: DESC Currently applied compensation
    '}
    fCurrentBacklash: LREAL;
END_STRUCT
END_TYPE

// ---- DUTs/ST_PositionState.TcDUT
TYPE ST_PositionState :
    // Defines settings and current safety status for moves to specific positions for an axis
STRUCT
    // Name as queried via the NAME PV in EPICS
    {attribute 'pytmc' := '
        pv: NAME
        io: input
        field: DESC Name of this position state
    '}
    sName: STRING := 'Invalid';

    // Position associated with this state
    {attribute 'pytmc' := '
        pv: SETPOINT
        io: io
        field: DESC Axis position associated with this state
        autosave_pass1: VAL
    '}
    fPosition: LREAL;

    {attribute 'pytmc' := '
        pv: ENCODER
        io: i
        field: DESC Encoder count associated with this state
    '}
    nEncoderCount: UDINT;

    // Maximum allowable deviation from fPosition while at the state
    fDelta: LREAL;

    // Speed at which to move to this state
    {attribute 'pytmc' := '
        pv: VELO
        io: io
        field: DESC Speed at which to move to this state
        autosave_pass1: VAL
    '}
    fVelocity: LREAL;

    // (optional) Acceleration to use for moves to this state
    fAccel: LREAL;

    // (optional) Deceleration to use for moves to this state
    fDecel: LREAL;

    // Safety parameter. This must be set to TRUE by the PLC program to allow moves to this state. This is expected to change as conditions change.
    {attribute 'pytmc' := '
        pv: MOVE_OK
        io: i
        field: ZNAM FALSE
        field: ONAM TRUE
        field: DESC TRUE if the move would be safe
    '}
    bMoveOk: BOOL;

    // Signifies to FB_PositionStateLock that this state should be immutable
    bLocked: BOOL;

    // Set this to TRUE when you make your state. This defaults to FALSE so that uninitialized states can never be moved to
    bValid: BOOL;

    // Set this to TRUE when you want to use the raw encoder counts to define the state
    bUseRawCounts: BOOL;

    // Is set to TRUE by FB_PositionStateInternal when called
    bUpdated: BOOL;

    // We give this a state name and it is used to load parameters from the pmps database.
    stPMPS: ST_DbStateParams;
END_STRUCT
END_TYPE

// ---- DUTs/E_EpicsMotorCmd.TcDUT
{attribute 'qualified_only'}
{attribute 'strict'}
TYPE E_EpicsMotorCmd :
    // Defines valid EPICS commands for nCommand
(
    JOG := 0,
    MOVE_VELOCITY := 1,
    MOVE_RELATIVE := 2,
    MOVE_ABSOLUTE := 3,
    MOVE_MODULO := 4,
    HOME := 10,
    GEAR := 30,
	CALIBRATE:=40
);
END_TYPE

// ---- POUs/Motion/DS402/I_DS402GenericDrive.TcIO
INTERFACE I_DS402GenericDrive

METHOD ExposedParameters
VAR_INPUT
	Enable : BOOL; 
    tRefreshDelay: TIME;
END_VAR
END_METHOD

METHOD Home
VAR_INPUT
    Enable 				: BOOL;
END_VAR
END_METHOD

METHOD ModeOperation
VAR_INPUT
END_VAR
END_METHOD

METHOD MoveAbsolute
VAR_INPUT
END_VAR
END_METHOD

METHOD PersistParameters
VAR_INPUT
	 Enable: BOOL;
END_VAR
END_METHOD

METHOD Power : BOOL
VAR_INPUT
END_VAR
END_METHOD

METHOD ReadDriveCodes : BOOL
END_METHOD

METHOD Reset : BOOL
VAR_INPUT
END_VAR
END_METHOD

METHOD RestoreMotionParams
VAR_INPUT
    Enable	: BOOL;
END_VAR
END_METHOD

METHOD ScaleDriveParams
VAR_INPUT
END_VAR
END_METHOD

METHOD ScaleEncRawValue
VAR_INPUT
END_VAR
END_METHOD

METHOD ScaleHomingParams
VAR_INPUT
END_VAR
END_METHOD

METHOD ScaleJogParams
VAR_INPUT
END_VAR
END_METHOD

METHOD SetChanParams
VAR_INPUT
    Enable : BOOL;
END_VAR
END_METHOD

METHOD SetEnables
VAR_INPUT
END_VAR
END_METHOD

METHOD SetEpicsStatus
VAR_INPUT
END_VAR
END_METHOD

METHOD SetJogParams
VAR_INPUT
	Enable : BOOL;
END_VAR
END_METHOD

METHOD StateMachine
VAR_INPUT
	Enable : BOOL;
END_VAR
END_METHOD

METHOD  StepMove
VAR_INPUT
	Enable : BOOL;
END_VAR
END_METHOD

METHOD WriteParameterNC
VAR_INPUT
    Execute:BOOL;
    ParameterNumber : MC_AxisParameter;
    ParameterValue	: LREAL;
END_VAR
END_METHOD

END_INTERFACE

// ---- POUs/Motion/DS402/FB_MotionStageE727.TcPOU
(*	MCS2 Motion Stage . Controller a stage in CSP (NC), STEP_MODE and Homing via DS402 interface
     Using an overriden Position Holding timer. power enable mode must be 'DURING_MOTION'. for close loop aka CSP control
    set bServo PV to true, fort open loop step mode bServo must be cleared
*)
{attribute 'call_after_init'}
FUNCTION_BLOCK FB_MotionStageE727 IMPLEMENTS I_DS402GenericDrive
VAR
    {attribute 'no_copy'}
    stMotionStage  : REFERENCE TO ST_MotionStage;
    // Hardware I/O
    stDS402Drive 		: ST_DS402Drive;
    // Must be Provided
    {attribute 'hide'}
    eModule 			: E_Module;
    {attribute 'hide'}
    eHomeMode			: E_EpicsHomeCmd :=E_EpicsHomeCmd.AUTOZERO;
    {attribute 'hide'}
    eBufferMode 		: MC_BufferMode := MC_BufferMode.MC_Aborting;
    {attribute 'hide'}
    eMotionState 		: E_MoveState;
    {attribute 'hide'}
    eHomeState  		: E_MoveState;
    {attribute 'hide'}
    fbMcPower 			: MC_Power;
    {attribute 'hide'}
    fbMcMoveAbsolute 	: MC_MoveAbsolute;
    {attribute 'hide'}
    fbMcHalt 			: MC_Halt;
    {attribute 'hide'}
    fbMcReset 			: MC_Reset;
    {attribute 'hide'}
    fbMcWriteParameter 	: MC_WriteParameter;
    {attribute 'hide'}
    fbMcReadParams		: MC_ReadParameterSet;
    {attribute 'hide'}
    bEnPosLag 			: BOOL;
    {attribute 'hide'}
    bWrongParameter 	: BOOL;
    {attribute 'hide'}
    bExecMove 			: BOOL;
    {attribute 'hide'}
    bExecHome 			: BOOL;
    {attribute 'hide'}
    bNewMoveReq 		: BOOL;
    {attribute 'hide'}
    bHomeBusy 			: BOOL;
    {attribute 'hide'}
    bPrepareDisable 	: BOOL;
    {attribute 'hide'}
    bStop  				: BOOL;
    {attribute 'hide'}
    bOperational  		: BOOL;
    {attribute 'hide'}
    bLimOverride  		: BOOL;
    // use this for motion time axis states
    {attribute 'hide'}
    bLocalExec			: BOOL;
    // Save abd restore encoder value
    {attribute 'hide'}
    bInit				: BOOL;
    {attribute 'hide'}
    bHomeDone 			: BOOL;
    {attribute 'hide'}
    bHomeModeEnabled	: BOOL;
    {attribute 'hide'}
    bCSPModeEnabled		: BOOL;
    {attribute 'hide'}
    bRestoreLoad		: BOOL;
    {attribute 'hide'}
    bExecParamsRead		: BOOL;
    {attribute 'hide'}
    bCommandMoveAbsolute : BOOL;
    {attribute 'hide'}
    bRecentEnPosLagStatus 	: BOOL;
    {attribute 'hide'}
    bHomeAborted : BOOL;
    {attribute 'hide'}
    bDS402ManualEnabled : BOOL;
    {attribute 'hide'}
    fMeasuredVelo		: LREAL;
    {attribute 'hide'}
    fMeasuredAcc		: LREAL;
    {attribute 'hide'}
    fScalingFactor		: LREAL:= 0.000001;
    {attribute 'hide'}
    fParameterValue : LREAL;
    {attribute 'hide'}
    fMeasuredPos 		: LREAL;
    {attribute 'hide'}
    nSoftLimMin     	: LINT;
    {attribute 'hide'}
    nSoftLimMax     	: LINT;
    {attribute 'hide'}
    tonSyncHoming 		: TON;
    {attribute 'hide'}
    tonSlowParamReadTimer: TON;
    {attribute 'hide'}
    NCParamsTimer 		: TON;
    {attribute 'hide'}
    tonRestoreRetry		: TON;
    {attribute 'hide'}
    rtAborted 			: R_TRIG;
    {attribute 'hide'}
    rtStopDone			: R_TRIG;
    {attribute 'hide'}
    rtExec 				: R_TRIG;
    {attribute 'hide'}
    rtMoveCmdShortcut 	: R_TRIG;
    {attribute 'hide'}
    rtHomeCmdShortcut 	: R_TRIG;
    {attribute 'hide'}
    rtEnableMode    	: R_TRIG;
    {attribute 'hide'}
    rtUserExec      	: R_TRIG;
    {attribute 'hide'}
    rtModeChange      	: R_TRIG;
    {attribute 'hide'}
    rtMoveDone    		: R_TRIG;
    {attribute 'hide'}
    {attribute 'hide'}
    rtNewMoveReq  		: R_TRIG;
    {attribute 'hide'}
    ftExec      		: F_TRIG;
    {attribute 'hide'}
    rtHomeDone 			: R_TRIG;
    {attribute 'hide'}
    rtCSPModeOk			: R_TRIG;
    {attribute 'hide'}
    rtHomeModeEnable	: R_TRIG;
    {attribute 'hide'}
    nSubIndex			: BYTE := 0;
    {attribute 'hide'}
    nChanSoftwareLimIdx : WORD;
    {attribute 'hide'}
    nChanErrorCodeIdx 	: WORD;
    {attribute 'hide'}
    nChanSoftLimitIdx 	: WORD;
    {attribute 'hide'}
    bLocalReset: BOOL;
    {attribute 'hide'}
    nCommandLocal: INT := 3;
    {attribute 'hide'}
    nCmdDataLocal: INT;

END_VAR

VAR CONSTANT
    {attribute 'hide'}
    nChanSoftLimitBase	: WORD := 16#607D;
    {attribute 'hide'}
    nErrorCodeBase  	: WORD := 16#603F;
    // this true for SmartAct MCS2 and E-727.
    {attribute 'hide'}
    nChanOfsBase		: WORD := 16#800;

END_VAR

VAR PERSISTENT
    bSaved	: BOOL;
    fSavedPosition	: LREAL;
END_VAR

IF NOT __ISVALIDREF(stMotionStage) THEN
    RETURN;
END_IF

(* Done once after init*)
IF bInit THEN
    stMotionStage.nMotionAxisID := stMotionStage.Axis.NcToPlc.AxisId;
    (* Clear drive error/wraning condition, in open loop mode
       this will trigger a correct startup for procedure *)
    stDS402Drive.nDS402DriveControl := 128;
    // fist cycle reading of NC paramters
    bExecParamsRead := TRUE;
    bInit := FALSE;
END_IF
(* Check for the plc shortcut commands
   Used for testing or to circumvent motor record issues*)
rtMoveCmdShortcut(CLK:=stMotionStage.bMoveCmd);
rtHomeCmdShortcut(CLK:=stMotionStage.bHomeCmd);

(* Execute on rising edge*)
IF rtMoveCmdShortcut.Q AND NOT stMotionStage.bExecute THEN
    stMotionStage.bExecute:=TRUE;
    stMotionStage.nCommand := E_EpicsMotorCmd.MOVE_ABSOLUTE;
    bEnPosLag := bRecentEnPosLagStatus;
    fParameterValue := BOOL_TO_LREAL(bRecentEnPosLagStatus);

ELSIF rtHomeCmdShortcut.Q AND NOT stMotionStage.bExecute THEN
    stMotionStage.bExecute:= NOT ( stMotionStage.nCmdData=E_EpicsHomeCmd.ABSOLUTE_SET )
                            OR NOT ( stMotionStage.nCmdData=E_EpicsHomeCmd.NONE);
    stMotionStage.nCommand:=E_EpicsMotorCmd.HOME;
    (* Automatically fill the correct nCmdData for homing*)
    stMotionStage.nCmdData:=stMotionStage.nHomingMode;
    (*	Positional lag is not evaluated by E727 during homing, but NC does evaluated
        the condition which will lead to error as the lag is significant during homing
        disable the NC lag check and reenable it after homing is done
    *)
    IF stMotionStage.stAxisParameters.bCtrlEnablePosDiffControl.0 THEN
        bRecentEnPosLagStatus := stMotionStage.stAxisParameters.bCtrlEnablePosDiffControl.0;
        bEnPosLag := TRUE;
        fParameterValue := 0;
    END_IF

END_IF

(* entry point for local and EPICS main execs *)
rtUserExec(CLK:=stMotionStage.bExecute);
(* if a Move/Home Goal is comfirmed and there is no persistant
   error conditions, then we have a valid move request.*)
bNewMoveReq S= NOT stMotionStage.bBusy AND rtUserExec.Q AND NOT stMotionStage.bError;
(* this Move request is valid till an error occurs or the currently move is done *)
bNewMoveReq R= NOT stMotionStage.bExecute OR stMotionStage.bError;
bPrepareDisable R= bNewMoveReq;
rtNewMoveReq(CLK:=bNewMoveReq);
(* Moves are automatically allowed if no safety hooks.
   Otherwise, some other code will set this.*)
stMotionStage.bSafetyReady S= stMotionStage.bPowerSelf;
(* Set the proper command for the request move;
   if bservo not set, manual step moves will be performed *)
IF rtUserExec.Q THEN
    // Transfer nCommand and nCmdData to local copies at rising edge of bExecute (avoid issues if nCommand or nCmdData are changed during a command)
    nCmdDataLocal:=stMotionStage.nCmdData;
    nCommandLocal:=stMotionStage.nCommand;
    (* attempting to move an axis without homing first? *)
    IF stMotionStage.nHomingMode <> E_EpicsHomeCmd.NONE AND NOT stMotionStage.bHomed THEN
        (* one can just set bHome here even though no homing was done?*)
        stMotionStage.sErrorMessage:='Axis homing mode set, but homing routine pending';
    END_IF
END_IF

(* Set the drive in the correct operating mode. based on requested move command!
    NB: bservo must set for close loop motion
*)
ModeOperation();

(* NB: This is the only tested mode of operation so far. also aligned
    piezo drive position holding feature
*)
rtEnableMode(CLK:=(stMotionStage.nEnableMode = E_StageEnableMode.DURING_MOTION));
(* Handle auto-enable timing *)
CASE stMotionStage.nEnableMode OF
    (* Not recommended, not tested *)
    E_StageEnableMode.ALWAYS:
        stMotionStage.bEnable:=TRUE;
    E_StageEnableMode.DURING_MOTION:
        IF rtEnableMode.Q THEN
            stMotionStage.bEnable := FALSE;
        END_IF
        IF rtNewMoveReq.Q THEN
            (*MC block are not compatible with open loop Motion
                thus we wathc for correct close loop modes to use NC features *)
            stMotionStage.bEnable S= stMotionStage.bSafetyReady;
            bStop:=FALSE;
        END_IF
END_CASE
(*	Interlock mainly react on internal limit conditions inthe ove direction.
    MCS2 drive will go into error state when an internal limit is hit *)
Interlock();

IF bCSPModeEnabled THEN
    (*CSP using TwinCAT NC*)
    bLocalExec:= NOT stMotionStage.bError AND stMotionStage.bExecute AND stMotionStage.bAllEnable AND stMotionStage.bEnableDone AND stMotionStage.bSafetyReady;
ELSIF bHomeModeEnabled THEN
    bLocalExec:= NOT stMotionStage.bError AND stMotionStage.bExecute AND stMotionStage.bAllEnable AND  bOperational AND  stMotionStage.bSafetyReady;
ELSE
    bLocalExec:= FALSE;
END_IF

bExecHome:=bLocalExec AND stMotionStage.nCommand = 10;
bExecMove:=bLocalExec AND NOT bExecHome;

(* When we start, set the busy/done appropriately
   NB: CLose loop control using NC *)
rtExec(CLK:=bLocalExec);
IF rtExec.Q THEN
    // Release previous interruption if any
    stDS402Drive.nDS402DriveControl.8 := FALSE;
    stMotionStage.bDone := FALSE;
END_IF

(* updated axis status
   Not needed in manual mode *)
IF NOT bDS402ManualEnabled THEN
    stMotionStage.Axis.ReadStatus();
END_IF

(* Get a definitive bEnabled reading
   NB: use only in close loop mode, NC feature needed*)
CASE stMotionStage.Axis.Status.MotionState OF
    (* We are not enabled if there is an issue*)
    MC_AXISSTATE_UNDEFINED, MC_AXISSTATE_DISABLED, MC_AXISSTATE_ERRORSTOP:
        stMotionStage.bEnableDone := FALSE;
    ELSE
        stMotionStage.bEnableDone := TRUE;
END_CASE
//
IF stMotionStage.bReset THEN
    stMotionStage.bExecute:=FALSE;
    stMotionStage.bError := FALSE;
    stMotionStage.nErrorId := 0;
    stMotionStage.sErrorMessage:='';
    stMotionStage.sCustomErrorMessage:='';
    (*Manual Drive reset*)
    IF bDS402ManualEnabled THEN
        stDS402Drive.nDS402DriveControl := 128;
    ELSE
        bLocalReset := TRUE;
    END_IF

    stMotionStage.bReset:=FALSE;
END_IF

// Halt is always a user stop during motion
bStop S= NOT bLocalExec AND ((bHomeBusy AND (nCommandLocal=10)) OR (fbMcMoveAbsolute.Busy AND (nCommandLocal=3)));

//auto handle position lag monitoring, disable during homing.
WriteParameterNC(	Execute:=bEnPosLag,
                    ParameterNumber:=MC_AxisParameter.AxisEnPositionLagMonitoring,
                    ParameterValue:=fParameterValue);

(* Requested commands processing *)
CASE nCommandLocal OF
    E_EpicsMotorCmd.MOVE_ABSOLUTE:
        (*NC CSP Move Handling*)
        (* Trigger MC_Reset for close loop operation aka CSP mode *)
        Reset();
        Power();
        Halt();
        (*Wait for drive to be in the correct mode after a request was validated *)
        bCommandMoveAbsolute := bExecMove AND fbMcPower.Status AND bCSPModeEnabled;
        MoveAbsolute();
        (*IN CSP mode the drive control word is update via the NC
          Manual step mode and Homing will override this *)
         stDS402Drive.nDS402DriveControl := stDS402Drive.nDS402DriveControlNC;
    E_EpicsMotorCmd.HOME:
        (*DS402 Manual Homing*)
       Home(Enable:=TRUE);
END_CASE

stMotionStage.bBusy := bHomeBusy OR fbMcMoveAbsolute.Busy;

(* Check done moving via user stop, limit hit, Target Position reached, or from homing.*)
rtMoveDone(CLK:=fbMcMoveAbsolute.Done);
rtHomeDone(CLK:=bHomeDone);
rtStopDone(CLK:=fbMcHalt.Done);
rtAborted(CLK:=bHomeAborted);
IF rtAborted.Q OR rtStopDone.Q OR rtMoveDone.Q OR rtHomeDone.Q THEN
    IF NOT stMotionStage.bDone THEN
        stMotionStage.bHomed := bHomeDone;
        stMotionStage.bExecute:=FALSE;
        bCommandMoveAbsolute := FALSE;
        stMotionStage.bDone := fbMcMoveAbsolute.Done OR bHomeDone;
        IF bDS402ManualEnabled THEN
            // No standstill in Manual Mode
            stMotionStage.bEnable:=FALSE;
            (*Restore Postional lag monitoring*)
            bEnPosLag := FALSE;
        END_IF
        (* Release the internal limit override*)
        bLimOverride := FALSE;
        bHomeAborted := FALSE;
    END_IF
END_IF

(* updated axis status
   Not needed in manual mode *)
IF NOT bDS402ManualEnabled THEN
    stMotionStage.Axis.ReadStatus();
END_IF

ftExec(CLK:=stMotionStage.bExecute);
(*Handle auto-disable timing*)
bPrepareDisable S= stMotionStage.nEnableMode = E_StageEnableMode.DURING_MOTION AND ftExec.Q;
(* Delay the disable until we reach standstill *)
IF bPrepareDisable AND stMotionStage.Axis.Status.StandStill THEN
    bPrepareDisable:=FALSE;
    stMotionStage.bEnable:=FALSE;
END_IF

(* update encoder value and calibrated position*)
ScaleEncRawValue();
(*Drive parameters*)
ExposedParameters(Enable:=TRUE, tRefreshDelay:=T#2S);
(*Sync NC setting to drive settings*)
UpdateDriveMonitoringParams(Enable:=stMotionStage.bAxisParamsInit AND NOT stMotionStage.bBusy);
(* Save and restore as long as not an absolute encoder*)
PersistParameters( Enable:=stMotionStage.nHomingMode <> E_EpicsHomeCmd.NONE);
(*Restore encoder value at initialization*)
RestoreMotionParams(Enable:=stMotionStage.nHomingMode <> E_EpicsHomeCmd.NONE);

(*EPICS Motor record Update*)
UpdateEpicsStatus();
(*
    Error from functions and Nc. The error will send to EPICS interface based on predifined
    priority: axis, power, backlash, absoluteMove, etc...
*)
IF fbMcPower.Error AND fbMcPower.Active THEN
    stMotionStage.bError:=fbMcPower.Error;
    stMotionStage.nErrorId:=fbMcPower.ErrorID;
ELSIF fbMcMoveAbsolute.Error THEN
    stMotionStage.bError:=fbMcMoveAbsolute.Error;
    stMotionStage.nErrorId:=fbMcMoveAbsolute.ErrorID;
ELSIF fbMcHalt.Error AND fbMcHalt.Active THEN
    stMotionStage.bError:=fbMcHalt.Error;
    stMotionStage.nErrorId:=fbMcHalt.ErrorID;
ELSIF fbMcReset.Error  THEN
    stMotionStage.bError:=fbMcReset.Error;
    stMotionStage.nErrorId:=fbMcReset.ErrorID;
ELSIF fbMcWriteParameter.Error THEN
    stMotionStage.bError:=fbMcWriteParameter.Error;
    stMotionStage.nErrorId:=fbMcWriteParameter.ErrorID;
ELSIF fbMcReadParams.Error AND NOT stMotionStage.bBusy THEN
    stMotionStage.bError:=fbMcReadParams.Error;
    stMotionStage.nErrorId:=fbMcReadParams.ErrorID;
ELSE
    IF stMotionStage.bBusy THEN
        stMotionStage.sErrorMessage := '';
        stMotionStage.sCustomErrorMessage := '';
    END_IF
END_IF;

(*Double function, prioritize NC error otherwise read drive channel error code*)
ReadDriveCodes();

IF stMotionStage.sCustomErrorMessage <> ''
    AND stMotionStage.sErrorMessage = '' THEN
    stMotionStage.sErrorMessage := stMotionStage.sCustomErrorMessage;
END_IF

(*Clear motion flag when error occurs*)
IF stMotionStage.bError  THEN
    stMotionStage.bBusy := FALSE;
    stMotionStage.bDone := FALSE;
    stMotionStage.bEnable := FALSE;
END_IF

(* We've got the rising edge clear this flags.*)
stMotionStage.bMoveCmd:=FALSE;
stMotionStage.bHomeCmd:=FALSE;

METHOD PUBLIC  ExposedParameters
VAR_INPUT
    Enable : BOOL;
    tRefreshDelay: TIME;
END_VAR
// Periodic update of NC parameters
NCParamsTimer( IN:=Enable AND NOT bExecParamsRead, PT:=tRefreshDelay);
bExecParamsRead S= NCParamsTimer.Q;
fbMcReadParams(
    Parameter:=stMotionStage.stAxisParameters,
    Axis:=stMotionStage.Axis,
    Execute:= bExecParamsRead );

// Copy axis parameters that we want to expose to the EPICS layer.
stMotionStage.stAxisParametersExposed.bCtrlEnablePosDiffControl     := stMotionStage.stAxisParameters.bCtrlEnablePosDiffControl;
stMotionStage.stAxisParametersExposed.bEncEnableSoftEndMaxControl   := stMotionStage.stAxisParameters.bEncEnableSoftEndMaxControl;
stMotionStage.stAxisParametersExposed.bEncEnableSoftEndMinControl   := stMotionStage.stAxisParameters.bEncEnableSoftEndMinControl;
stMotionStage.stAxisParametersExposed.fAccelerationMax              := stMotionStage.stAxisParameters.fAccelerationMax;
stMotionStage.stAxisParametersExposed.fCtrlPosDiffMax               := stMotionStage.stAxisParameters.fCtrlPosDiffMax;
stMotionStage.stAxisParametersExposed.fCtrlPosDiffMaxTime           := stMotionStage.stAxisParameters.fCtrlPosDiffMaxTime;
stMotionStage.stAxisParametersExposed.fDecelerationMax              := stMotionStage.stAxisParameters.fDecelerationMax;
stMotionStage.stAxisParametersExposed.fEncSoftEndMax                := stMotionStage.stAxisParameters.fEncSoftEndMax;
stMotionStage.stAxisParametersExposed.fEncSoftEndMin                := stMotionStage.stAxisParameters.fEncSoftEndMin;
stMotionStage.stAxisParametersExposed.fVeloMaximum                  := stMotionStage.stAxisParameters.fVeloMaximum;
stMotionStage.stAxisParametersExposed.fEncOffset               		:= stMotionStage.stAxisParameters.fEncOffset;
stMotionStage.stAxisParametersExposed.fEncScaleFactorInternal       := stMotionStage.stAxisParameters.fEncScaleFactorInternal;

bExecParamsRead R= fbMcReadParams.Done OR fbMcReadParams.Error;
stMotionStage.bAxisParamsInit S= fbMcReadParams.Done;
END_METHOD

//FB_Init is always available implicitly and it is used primarily for initialization.
//The return value is not evaluated. For a specific influence, you can also declare the
//methods explicitly and provide additional code there with the standard initialization
//code. You can evaluate the return value.
METHOD FB_Init: BOOL
VAR_INPUT
    bInitRetains: BOOL; // TRUE: the retain variables are initialized (reset warm / reset cold)
    bInCopyCode: BOOL;  // TRUE: the instance will be copied to the copy code afterward (online change)
    stPiezoStage		:	REFERENCE TO ST_MotionStage;
    (*Mandatory must be unique for each MCS2 axis *)
    eModule : E_Module;
END_VAR
THIS^.stMotionStage REF= stPiezoStage;
THIS^.eModule := eModule;
END_METHOD

METHOD Halt : BOOL
fbMcHalt(
    Axis := stMotionStage.Axis,
    Execute := bStop AND bCSPModeEnabled,
    Deceleration := stMotionStage.fDeceleration,
    BufferMode := eBufferMode,
);
END_METHOD

METHOD PUBLIC Home
VAR_INPUT
    Enable 				: BOOL;
END_VAR
VAR_INST
    {attribute 'hide'}
    bMove 				: BOOL;
END_VAR
CASE eHomeMode OF
    E_EpicsHomeCmd.AUTOZERO:
        bMove S=  bExecHome;
    E_EpicsHomeCmd.NONE:
        bMove := FALSE;
        bHomeBusy :=  bExecHome;
        bHomeDone := NOT  bExecHome;
    ELSE
        bMove := FALSE;
END_CASE

IF bMove THEN
    CASE eHomeState OF
        // Wait for a rising edge
        E_MoveState.IDLING:
            IF bHomeModeEnabled AND bExecHome THEN
                bHomeDone := FALSE;
                bHomeBusy := TRUE;
                stMotionStage.bDone := FALSE;
                stDS402Drive.nDS402DriveControl:=15;
                eHomeState :=  E_MoveState.INIT;
            END_IF
        E_MoveState.INIT:
                        stDS402Drive.nDS402DriveControl.4:=1;
                                        eHomeState := E_MoveState.STARTED;
        E_MoveState.STARTED :
            // this is a comfirmation that routine is ongoing
            IF NOT stDS402Drive.stDS402DriveStatus.TargetReached
                AND NOT stDS402Drive.stDS402DriveStatus.Bit13_OpModeSpecific THEN
                bHomeBusy:=TRUE;
                bHomeDone:=FALSE;

                eHomeState:=E_MoveState.IN_PROGRESS;
            END_IF

        E_MoveState.IN_PROGRESS :

        IF bStop THEN
         stDS402Drive.nDS402DriveControl.8 :=1;
          bHomeAborted := TRUE;
          eHomeState:=E_MoveState.INTERRUPTED;

        // Genral Motion error i.e Following error ?
        ELSIF stDS402Drive.stDS402DriveStatus.Bit13_OpModeSpecific
                OR stDS402Drive.stDS402DriveStatus.WarningCondition THEN
            stMotionStage.bError := TRUE;
            eHomeState:=E_MoveState.ERROR;

        // Reached
        ELSIF stDS402Drive.stDS402DriveStatus.TargetReached
            AND stDS402Drive.stDS402DriveStatus.Bit12_OpModeSpecific
            AND NOT stDS402Drive.stDS402DriveStatus.Bit13_OpModeSpecific THEN
           eHomeState:=E_MoveState.DONE;
        END_IF
        E_MoveState.INTERRUPTED:
            bHomeBusy:=FALSE;
            eHomeState:=E_MoveState.IDLING;
        E_MoveState.DONE:
            bHomeBusy:=FALSE;
            bHomeDone:=TRUE;
            stMotionStage.fPosition:=0.0;

            IF (stMotionStage.nEnableMode = E_StageEnableMode.DURING_MOTION ) THEN
                stDS402Drive.nDS402DriveControl.4:=FALSE;

            ELSE
                stDS402Drive.nDS402DriveControl:=6;
            END_IF
            eHomeState:=E_MoveState.IDLING;
        E_MoveState.ERROR:
            bHomeDone:=FALSE;
            bHomeBusy:= FALSE;
            IF bWrongParameter THEN
                stMotionStage.sCustomErrorMessage:='Invalid motion Parameters';
                bWrongParameter := FALSE;
                stMotionStage.bError := TRUE;
            END_IF
            IF NOT stMotionStage.bError THEN
                eHomeState:=E_MoveState.IDLING;
            END_IF
    END_CASE
END_IF
END_METHOD

METHOD PUBLIC Interlock

VAR_INST
    {attribute 'hide'}
    bPositiveDirection  : BOOL;
    {attribute 'hide'}
    bNegativeDirection  : BOOL;
    {attribute 'hide'}
    ftForwardEnabled  	: F_TRIG;

    {attribute 'hide'}
    ftBackwardEnabled 	: F_TRIG;
END_VAR
// Positive or Negative direction
bPositiveDirection:=stMotionStage.bBusy AND stMotionStage.fPosDiff > 0;
bNegativeDirection:=stMotionStage.bBusy AND stMotionStage.fPosDiff < 0;

// For SmartAct MCS2 these limit are range and enstop limits. however a single bit in the status is used
// bLimOverride  : act as an override after limit was hit to allow reverse movement
stMotionStage.bLimitForwardEnable :=  bLimOverride OR NOT( bPositiveDirection AND stDS402Drive.stDS402DriveStatus.InternalLimitActive );
stMotionStage.bLimitBackwardEnable := bLimOverride OR NOT( bNegativeDirection AND stDS402Drive.stDS402DriveStatus.InternalLimitActive );

// use falling trigger to avoid spaming  sErrorMessage
ftForwardEnabled(CLK:=stMotionStage.bLimitForwardEnable);
ftBackwardEnabled(CLK:=stMotionStage.bLimitBackwardEnable);

IF  NOT bHomeBusy AND ftForwardEnabled.Q THEN
    // Not an error, just a warning
    stMotionStage.sCustomErrorMessage:='Cannot move past positive limit.';
    bLimOverride := TRUE;
END_IF

IF NOT bHomeBusy AND ftBackwardEnabled.Q THEN
    // Not an error, just a warning
    stMotionStage.sCustomErrorMessage:='Cannot move past Negative limit.';
    bLimOverride := TRUE;
END_IF

IF NOT stMotionStage.bError AND stMotionStage.bExecute AND NOT stMotionStage.bUserEnable THEN
    stMotionStage.bError := TRUE;
    stMotionStage.nErrorId := 1;
    stMotionStage.sCustomErrorMessage := 'Move requested, but user enable is disabled!';
END_IF

// Update all enable booleans
SetEnables();
END_METHOD

(*Switch the drive mod eof Operation
  Servo On: Profil Positioning or HOME
  Servo Off : STEP mode
*)
METHOD ModeOperation

VAR_INST
    tonSwitching : TON;
    bManualTransition: BOOL;
END_VAR
rtCSPModeOk(CLK:=( stDS402Drive.nModeOfOperationDisplay=E_DS402OpMode.CSP));
rtHomeModeEnable(CLK:=( stDS402Drive.nModeOfOperationDisplay=E_DS402OpMode.HOME));
// transition to close loop mode
IF rtCSPModeOk.Q THEN
    bHomeModeEnabled := FALSE;
    bCSPModeEnabled := TRUE;
ELSIF rtHomeModeEnable.Q THEN
    bHomeModeEnabled := TRUE;
    bCSPModeEnabled := FALSE;
    stDS402Drive.nDS402DriveControl := 0;
END_IF

IF rtUserExec.Q AND stMotionStage.bHomeCmd THEN
    IF (stDS402Drive.nModeOfOperationDisplay<>E_DS402OpMode.HOME) THEN
        stDS402Drive.nModeOfOperation := E_DS402OpMode.HOME;
        stDS402Drive.nDS402DriveControl := 128;
        // clear previous operational from switching away from this mode.
        bOperational := FALSE;
        bCSPModeEnabled := FALSE;
        bManualTransition := TRUE;
    ELSE
        bHomeModeEnabled := TRUE;
    END_IF
ELSIF rtUserExec.Q THEN
    IF (stDS402Drive.nModeOfOperationDisplay<>E_DS402OpMode.CSP) THEN
        stDS402Drive.nModeOfOperation := E_DS402OpMode.CSP;
        stDS402Drive.nDS402DriveControl := 128;
        bHomeModeEnabled := FALSE;
        bManualTransition := FALSE;
    ELSE
        bCSPModeEnabled := TRUE;
    END_IF
END_IF

bDS402ManualEnabled :=bHomeModeEnabled;
(*Handle correct startup procedure for manual move*)
StateMachine(Enable:=1);
END_METHOD

METHOD PUBLIC  MoveAbsolute

fbMcMoveAbsolute(
    Axis := stMotionStage.Axis,
    Execute := bCommandMoveAbsolute,
    Position := stMotionStage.fPosition,
    Velocity := stMotionStage.fVelocity,
    Acceleration := stMotionStage.fAcceleration,
    Deceleration := stMotionStage.fDeceleration,
    BufferMode := eBufferMode,
);
END_METHOD

METHOD PersistParameters
VAR_INPUT
    Enable	: BOOL;
END_VAR

VAR_INST
    {attribute 'hide'}
    bEncError			: BOOL;

    {attribute 'hide'}
    bRestoreWaitRetry	: BOOL;
END_VAR
// Save Encoder position
// needs some pre-conditions to use persistent storage
IF Enable THEN
    // Check ST_MotionStage for an encoder error (range 0x44nn)
    bEncError:= stMotionStage.Axis.Status.Error AND  ( stMotionStage.Axis.Status.ErrorID  >= 16#4400  AND stMotionStage.Axis.Status.ErrorID <= 16#44FF );
    // Do not save if we're currently loading or if there is an encoder error
    IF NOT bRestoreLoad AND NOT bEncError AND NOT bRestoreWaitRetry THEN
        fSavedPosition := stMotionStage.Axis.NcToPlc.ActPos;
        // This persistent variable lets us check if anything was saved
        // It will be TRUE at startup if we have saved values
        bSaved := TRUE;
        (*
            use this with a timer of a change threshold on the fActPosition
            to trigger a save from this PLC program. otherwise this will be a spamming
            persistence, filling up the disk.
        *)
        //iPersistentDataStorage.TriggerWriteOfPersistentData := bSaveEnabled;
    END_IF
END_IF
END_METHOD

{attribute 'call_after_init'}
(*	eModule: Mandatory must be unique for each MCS2 axis
    clears startup errors or warnings. the process is completed at run time
    SDO update of Drive and open Loop parameter Indexes based on module number
*)
METHOD PostInit
VAR_INPUT
END_VAR
(* SDO update of Drive and open Loop parameter Indexes based on module number*)
nChanErrorCodeIdx	:= nErrorCodeBase		+ ((eModule-1) * nChanOfsBase);
nChanSoftLimitIdx	:= nChanSoftLimitBase 	+ ((eModule-1) * nChanOfsBase);
bInit := TRUE;
END_METHOD

METHOD Power : BOOL
fbMcPower(
    Axis := stMotionStage.Axis,
    Enable := stMotionStage.bAllEnable AND bCSPModeEnabled,
    Enable_Positive := stMotionStage.bAllForwardEnable,
    Enable_Negative := stMotionStage.bAllBackwardEnable,
    Override := 100.0,
    BufferMode := eBufferMode );
END_METHOD

(* Read Drive error codes after a motion or fault condition occured *)
METHOD ReadDriveCodes : BOOL
VAR_INST
    {attribute 'hide'}
    fbErrorRead			: FB_EcCoESdoRead;
    {attribute 'hide'}
    nPiezoErrorCode   	: UDINT;
    {attribute 'hide'}
    fbLogError  		: FB_LogMotionError;
    {attribute 'hide'}
    ftErrorReadDone  	: F_TRIG;
END_VAR
fbErrorRead( sNetId:= THIS^.stMotionStage.stAxisParameters.sAmsNetId,
             nSlaveAddr:=stDS402Drive.nSlaveAddr,
             nIndex:=nChanErrorCodeIdx,
             nSubIndex :=nSubIndex,
             pDstBuf:= ADR(nPiezoErrorCode),
             cbBufLen:=SIZEOF(nPiezoErrorCode),
             bExecute:= stMotionStage.bError );

ftErrorReadDone(CLK:=fbErrorRead.bBusy);
IF ftErrorReadDone.Q THEN
    IF 	NOT fbErrorRead.bError AND nPiezoErrorCode <> 0 THEN
        stMotionStage.nErrorId := nPiezoErrorCode;
    END_IF
    stMotionStage.sErrorMessage := F_MotionErrorCodeLookup(nErrorId:=stMotionStage.nErrorId);
    fbLogError( stMotionStage:=stMotionStage, bEnable:=stMotionStage.bError);
END_IF
END_METHOD

METHOD Reset : BOOL
fbMcReset(
    Axis := stMotionStage.Axis,
    Execute := bLocalReset AND bCSPModeEnabled
);

IF fbMcReset.Done OR fbMcReset.Error THEN
    bLocalReset := FALSE;
END_IF
END_METHOD

METHOD RestoreMotionParams
VAR_INPUT
    Enable	: BOOL;
END_VAR

VAR_INST
    {attribute 'hide'}
    fbSetPos			: MC_SetPosition;
    {attribute 'hide'}
    bLoad				: BOOL;
    {attribute 'hide'}
    bRestoreDone 		: BOOL;
    {attribute 'hide'}
    bRestoreInit		: BOOL;
    {attribute 'hide'}
    bRestoreWaitRetry	: BOOL;
    {attribute 'hide'}
    nMaxRetries			: UINT := 10;
    {attribute 'hide'}
    nCurrTries			: UINT := 0;
    {attribute 'hide'}
    nLatchError			: UDINT;
END_VAR
IF Enable THEN
    // Trigger a load if anything was saved at all
    IF NOT bRestoreInit THEN
        bRestoreInit := TRUE;
        bRestoreLoad S= bSaved;
        fbSetPos.Options.ClearPositionLag := TRUE;
    END_IF

    // Set our position if bRestoreLoad is true
    fbSetPos( Axis:=stMotionStage.Axis, Execute:=bRestoreLoad, Position:=fSavedPosition);

    // Only load once, at startup
    bRestoreLoad R= fbSetPos.Done OR fbSetPos.Error;

    IF fbSetPos.Error THEN
        // Keep the error latched, it can disappear if Execute is set to FALSE
        nLatchError := fbSetPos.ErrorID;
        nCurrTries := nCurrTries + 1;
        IF nCurrTries >= nMaxRetries THEN
        // Alert the user that something has gone wrong
        stMotionStage.bError := TRUE;
        stMotionStage.nErrorId := nLatchError;
        stMotionStage.sCustomErrorMessage := 'Error loading previously saved position.';
        ELSE
            // Reset the FB for the next retry
            fbSetPos( Axis:=stMotionStage.Axis, Execute:=bRestoreLoad, Position:=fSavedPosition);
            // Try again
            bRestoreWaitRetry := TRUE;
        END_IF
    ELSE
        IF NOT bRestoreDone THEN
            stMotionStage.fPosition := fSavedPosition;
        END_IF
        bRestoreDone := TRUE;
    END_IF

    tonRestoreRetry( IN := bRestoreWaitRetry, PT := T#100MS);
    bRestoreLoad S= tonRestoreRetry.Q;
    bRestoreWaitRetry R= tonRestoreRetry.Q;
END_IF
END_METHOD

METHOD ScaleDriveParams
nSoftLimMax := LREAL_TO_DINT((stMotionStage.stAxisParameters.fEncSoftEndMax / MAX(stMotionStage.stAxisParameters.fEncScaleFactorInternal, fScalingFactor)));
nSoftLimMin := LREAL_TO_DINT((stMotionStage.stAxisParameters.fEncSoftEndMin / MAX(stMotionStage.stAxisParameters.fEncScaleFactorInternal, fScalingFactor)));
END_METHOD

METHOD ScaleEncRawValue
VAR_INPUT
  //  bEnable: BOOL;
END_VAR
(* SmartACT: The encoder count from the Piezo drive is not a raw count from the embeded actuator device
   we get a calibrated nm value. thus the use of abs() since this value is signed.
   PI: to be discovered *)
IF stMotionStage.nRawEncoderDINT <> 0 THEN
    stMotionStage.nEncoderCount:=DINT_TO_UDINT(ABS(stMotionStage.nRawEncoderDINT));
ELSE
    stMotionStage.nEncoderCount:=0;
END_IF

// calibrated encoder readback
fMeasuredPos:=stMotionStage.Axis.NcToPlc.ActPos;
fMeasuredVelo :=stMotionStage.Axis.NcToPlc.ActVelo;
fMeasuredAcc := stMotionStage.Axis.NcToPlc.ActAcc;
stMotionStage.fPosDiff:=stMotionStage.Axis.NcToPlc.PosDiff;
END_METHOD

(*Scale Home Move parameters*)
METHOD ScaleHomingParams
END_METHOD

(*Scaled Open Loop Step mode motion parameters*)
METHOD ScaleJogParams
VAR_INPUT
END_VAR
END_METHOD

{warning 'Add method implementation '}
METHOD SetChanParams
VAR_INPUT
    Enable	: BOOL;
END_VAR
END_METHOD

METHOD SetEnables
VAR_INPUT
END_VAR
stMotionStage.bAllForwardEnable:=stMotionStage.bLimitForwardEnable AND (stMotionStage.bGantryForwardEnable OR NOT stMotionStage.bGantryAxis) AND stMotionStage.stEPSForwardEnable.bEPS_OK;
stMotionStage.bAllBackwardEnable:=stMotionStage.bLimitBackwardEnable AND (stMotionStage.bGantryBackwardEnable OR NOT stMotionStage.bGantryAxis) AND stMotionStage.stEPSBackwardEnable.bEPS_OK;

stMotionStage.bAllEnable:=stMotionStage.bEnable AND stMotionStage.bHardwareEnable AND stMotionStage.stEPSPowerEnable.bEPS_OK;
stMotionStage.bAllEnable R= NOT stMotionStage.bUserEnable;
END_METHOD

{warning 'Add method implementation '}
METHOD SetEpicsStatus
END_METHOD

{warning 'Add method implementation '}
METHOD SetJogParams
VAR_INPUT
    Enable	: BOOL;
END_VAR
END_METHOD

METHOD StateMachine
VAR_INPUT
    Enable : BOOL;
END_VAR

VAR_INST
    rtFault: R_TRIG;
    {attribute 'hide'}
    bFault				: BOOL;
END_VAR
rtFault(CLK:=bFault);
(*switch on disable*)
IF NOT stDS402Drive.stDS402DriveStatus.ReadyToSwitchOn
    AND NOT stDS402Drive.stDS402DriveStatus.SwitchedOn
    AND NOT stDS402Drive.stDS402DriveStatus.OperationEnabled
    AND NOT stDS402Drive.stDS402DriveStatus.Fault
    AND stDS402Drive.stDS402DriveStatus.VoltageEnabled
    AND NOT stDS402Drive.stDS402DriveStatus.QuickStopActive
    AND  stDS402Drive.stDS402DriveStatus.SwitchOnDisabled THEN
        bOperational := FALSE;
        IF bDS402ManualEnabled AND NOT bStop  THEN
            THIS^.stDS402Drive.nDS402DriveControl := 6;
        END_IF
(*Ready to switch*)
ELSIF stDS402Drive.stDS402DriveStatus.ReadyToSwitchOn
    AND NOT stDS402Drive.stDS402DriveStatus.SwitchedOn
    AND NOT stDS402Drive.stDS402DriveStatus.OperationEnabled
    AND NOT stDS402Drive.stDS402DriveStatus.Fault
    AND stDS402Drive.stDS402DriveStatus.VoltageEnabled
    AND stDS402Drive.stDS402DriveStatus.QuickStopActive
    AND NOT stDS402Drive.stDS402DriveStatus.SwitchOnDisabled THEN
        bFault := FALSE;
        bOperational := FALSE;
        IF bDS402ManualEnabled AND NOT bStop  THEN
            THIS^.stDS402Drive.nDS402DriveControl := 7;
        END_IF
(*Switch on*)
ELSIF stDS402Drive.stDS402DriveStatus.ReadyToSwitchOn
    AND  stDS402Drive.stDS402DriveStatus.SwitchedOn
    AND NOT stDS402Drive.stDS402DriveStatus.OperationEnabled
    AND NOT stDS402Drive.stDS402DriveStatus.Fault
    AND stDS402Drive.stDS402DriveStatus.VoltageEnabled
    AND stDS402Drive.stDS402DriveStatus.QuickStopActive
    AND NOT stDS402Drive.stDS402DriveStatus.SwitchOnDisabled THEN
        bOperational := FALSE;
        IF bDS402ManualEnabled AND NOT bStop  THEN
            THIS^.stDS402Drive.nDS402DriveControl := 15;
        END_IF
(*Operation enbaled*)
ELSIF stDS402Drive.stDS402DriveStatus.ReadyToSwitchOn
    AND stDS402Drive.stDS402DriveStatus.SwitchedOn
    AND stDS402Drive.stDS402DriveStatus.OperationEnabled
    AND NOT stDS402Drive.stDS402DriveStatus.Fault
    AND stDS402Drive.stDS402DriveStatus.VoltageEnabled
    AND stDS402Drive.stDS402DriveStatus.QuickStopActive
    AND NOT stDS402Drive.stDS402DriveStatus.SwitchOnDisabled THEN
        THIS^.bOperational := TRUE;
(*Fault*)
ELSIF  NOT stDS402Drive.stDS402DriveStatus.ReadyToSwitchOn
    AND NOT stDS402Drive.stDS402DriveStatus.SwitchedOn
    AND NOT stDS402Drive.stDS402DriveStatus.OperationEnabled
    AND stDS402Drive.stDS402DriveStatus.Fault
    AND stDS402Drive.stDS402DriveStatus.VoltageEnabled
    AND NOT stDS402Drive.stDS402DriveStatus.QuickStopActive
    AND NOT stDS402Drive.stDS402DriveStatus.SwitchOnDisabled THEN
        bOperational := FALSE;
        bFault := TRUE;

ELSE
    bFault := FALSE;
    bOperational := FALSE;
END_IF

// wait for parameter init done at startup to read potential error from drive
stMotionStage.bError := bFault AND stMotionStage.bAxisParamsInit;
END_METHOD

{warning 'Add method implementation '}
METHOD StepMove
VAR_INPUT
    Enable	: BOOL;
END_VAR
END_METHOD

(*	Drive parameters update
    Mirror NC axis parameters configurations to those of MCS2 drive
    1- Following error
    2- Home Speeds
    3- Home Acceleration
    4- SoftLimits
*)
METHOD UpdateDriveMonitoringParams
VAR_INPUT
    Enable : BOOL;
END_VAR

VAR_INST
    {attribute 'hide'}
    fbSetFErrorWin		: FB_EcCoESdoWrite;
    {attribute 'hide'}
    fbSetSoftLimMin		: FB_EcCoESdoWrite;
    {attribute 'hide'}
    fbSetSoftLimMax		: FB_EcCoESdoWrite;
    {attribute 'hide'}
    fbSetHomeOffs 		: FB_EcCoESdoWrite;
    {attribute 'hide'}
    fbSetHomeVeloFast 	: FB_EcCoESdoWrite;
    {attribute 'hide'}
    fbSetHomeVeloSlow 	: FB_EcCoESdoWrite;
    {attribute 'hide'}
    fbSetHomeAcc		: FB_EcCoESdoWrite;
    {attribute 'hide'}
    nRecentSoftLimMax 	: LINT;
    {attribute 'hide'}
    nRecentSoftLimMin 	: LINT;
    {attribute 'hide'}
    nRecentHomeVeloFast : UDINT;
    {attribute 'hide'}
    nRecentHomeVeloSlow : UDINT;
    {attribute 'hide'}
    nRecentHomeAcc 		: UDINT;
    {attribute 'hide'}
    nRecentFErrWin		: DINT;
    {attribute 'hide'}
    nRecentHomeOffset 	: DINT;
    {attribute 'hide'}
    nHomeOffs			: DINT;
    {attribute 'hide'}
    ftFErrWinSetDone	: F_TRIG;

    {attribute 'hide'}
    ftSoftLimMaxSetDone	: F_TRIG;
    {attribute 'hide'}
    ftSoftLimMinSetDone	: F_TRIG;
    {attribute 'hide'}
    ftHomeVeloFastSetDone: F_TRIG;
    {attribute 'hide'}
    ftHomeAccSetDone	: F_TRIG;
    {attribute 'hide'}
    ftHomeOffsSetDone	: F_TRIG;
    {attribute 'hide'}
    ftHomeVeloSlowSetDone: F_TRIG;
END_VAR
IF Enable THEN

    (*	Drive parameters update
        Mirror NC axis parameters configurations to those of MCS2 drive
        1- Following error.
        2- SoftLimits
        3-Position Range
    *)
  // add some safety here for  0 div.
  ScaleDriveParams();

  fbSetSoftLimMin(
    sNetId     := THIS^.stMotionStage.stAxisParameters.sAmsNetId,
    nSlaveAddr := stDS402Drive.nSlaveAddr,
    nIndex     := nChanSoftLimitIdx,
    nSubIndex  := 1,
    pSrcBuf    := ADR(nSoftLimMin),
    cbBufLen   := SIZEOF(nSoftLimMin),
    bExecute   := NOT stMotionStage.bBusy AND (nSoftLimMin <> nRecentSoftLimMin)
  );
  fbSetSoftLimMax(
    sNetId     := THIS^.stMotionStage.stAxisParameters.sAmsNetId,
    nSlaveAddr := stDS402Drive.nSlaveAddr,
    nIndex     := nChanSoftLimitIdx,
    nSubIndex  := 2,
    pSrcBuf    := ADR(nSoftLimMax),
    cbBufLen   := SIZEOF(nSoftLimMax),
    bExecute   := NOT stMotionStage.bBusy AND (nSoftLimMax <> nRecentSoftLimMax)
    );

  ftSoftLimMaxSetDone(CLK:=fbSetSoftLimMax.bBusy);
  ftSoftLimMinSetDone(CLK:=fbSetSoftLimMin.bBusy);

    IF ftSoftLimMaxSetDone.Q OR ftSoftLimMinSetDone.Q  THEN
        IF fbSetSoftLimMin.bError THEN
           stMotionStage.bError := fbSetSoftLimMin.bError;
           stMotionStage.nErrorId := fbSetSoftLimMin.nErrId;
        ELSIF fbSetSoftLimMax.bError THEN
           stMotionStage.bError := fbSetSoftLimMax.bError;
           stMotionStage.nErrorId := fbSetSoftLimMax.nErrId;
        ELSE
           nRecentSoftLimMax := nSoftLimMax;
           nRecentSoftLimMin := nSoftLimMin;
        END_IF
        fbSetSoftLimMin.bExecute := FALSE;
        fbSetSoftLimMax.bExecute := FALSE;
    END_IF
END_IF
END_METHOD

METHOD UpdateEpicsStatus
VAR_INPUT
END_VAR
//////////////////////////////////////////////////////////////////
// Transfer NC parameter status to EPICS
//////////////////////////////////////////////////////////////////
stMotionStage.stAxisStatus.bEnable:=stMotionStage.bAllEnable;
stMotionStage.stAxisStatus.bEnabled:=stMotionStage.bEnableDone; // account for PowerEnable from power block
stMotionStage.stAxisStatus.bError:=stMotionStage.bError;
stMotionStage.stAxisStatus.bHomeSensor:=stMotionStage.bHome;
stMotionStage.stAxisStatus.bLimitBwd:=stMotionStage.bAllBackwardEnable;
stMotionStage.stAxisStatus.bLimitFwd:=stMotionStage.bAllForwardEnable;
stMotionStage.stAxisStatus.bReset:=stMotionStage.bReset;
stMotionStage.stAxisStatus.fAcceleration:=fMeasuredAcc;
stMotionStage.stAxisStatus.fActDiff:=stMotionStage.fPosDiff;
stMotionStage.stAxisStatus.fActPosition:=fMeasuredPos;
stMotionStage.stAxisStatus.fActVelocity:=fMeasuredVelo;
stMotionStage.stAxisStatus.fDeceleration:=fMeasuredAcc;
stMotionStage.stAxisStatus.fOverride:=THIS^.fbMcPower.Override;
stMotionStage.stAxisStatus.fPosition:=stMotionStage.fPosition;
stMotionStage.stAxisStatus.fVelocity:=stMotionStage.fVelocity;
stMotionStage.stAxisStatus.nCmdData:=INT_TO_UINT(stMotionStage.nCmdData);  //Or nCmdDataLocal
stMotionStage.stAxisStatus.nCommand:=INT_TO_UINT(stMotionStage.nCommand);  //Or nCommandLocal
stMotionStage.stAxisStatus.nErrorId:=stMotionStage.nErrorId;
stMotionStage.stAxisStatus.bBusy:=stMotionStage.bBusy;
stMotionStage.stAxisStatus.bHomed:=stMotionStage.bHomed;
stMotionStage.stAxisStatus.bExecute:=bLocalExec;
stMotionStage.stAxisStatus.nCommand:=3; // If this is not 3, the IOC stops updating positions during homing
END_METHOD

(*	MCS2 OL Step parameters update
    1- Step
    2- Step Amplitude
    3- StepFreq
*)
METHOD UpdateServoOffMotionParams
VAR_INPUT
    Enable : BOOL;
END_VAR
END_METHOD

METHOD WriteParameterNC
VAR_INPUT
    Execute:BOOL;
    ParameterNumber : MC_AxisParameter;
    ParameterValue	: LREAL;
END_VAR
(*Do not change a moving axis parameter*)
fbMcWriteParameter(	Axis:=stMotionStage.Axis,
                    Execute:=(Execute AND stMotionStage.Axis.Status.NotMoving),
                    ParameterNumber:=ParameterNumber,
                    Value:=ParameterValue
                  );

// Reset execute after when done successfull or after abort reset
// this way the done and error condition is latched till next move or global reset.
END_METHOD

END_FUNCTION_BLOCK

// ---- POUs/Motion/DS402/FB_MotionStageMCS2.TcPOU
(*
    MCS2 Motion Stage
    Controls a stage in CSP (NC), STEP_MODE, and Homing via DS402 interface.
    - Uses overridden Position Holding timer.
    - power enable mode must be 'DURING_MOTION' for closed-loop (CSP) control.
    - Set bServo PV to true for closed-loop, clear for open-loop (step mode).
*)

{attribute 'call_after_init'}
FUNCTION_BLOCK FB_MotionStageMCS2 IMPLEMENTS I_DS402GenericDrive

VAR
    {attribute 'no_copy'}
    stMotionStage            : REFERENCE TO ST_MCS2Stage;
    // Hardware I/O
    stDS402Drive             : ST_DS402Drive;
    {attribute 'hide'}
    eModule                  : E_Module;
    {attribute 'hide'}
    eHomeMode                : E_EpicsHomeCmd := E_EpicsHomeCmd.AUTOZERO;
    {attribute 'hide'}
    eBufferMode              : MC_BufferMode := MC_BufferMode.MC_Aborting;
    {attribute 'hide'}
    eStepState             : E_MoveState;
    {attribute 'hide'}
    eHomeState               : E_MoveState;
    {attribute 'hide'}
    eCalibrateState         : E_MoveState;

    {attribute 'hide'}
    fbMcPower             : MC_Power;
    {attribute 'hide'}
    fbMcMoveAbsolute      : MC_MoveAbsolute;
    {attribute 'hide'}
    fbMcHalt              : MC_Halt;
    {attribute 'hide'}
    fbMcReset             : MC_Reset;
    {attribute 'hide'}
    fbMcWriteParameter    : MC_WriteParameter;
    {attribute 'hide'}
    fbMcReadParams        : MC_ReadParameterSet;
    {attribute 'hide'}
    bLastHoltTimeOut      : BOOL;
    {attribute 'hide'}
    bEnPosLag             : BOOL;
    {attribute 'hide'}
    bWrongParameter       : BOOL;
    {attribute 'hide'}
    bExecMove             : BOOL;
    {attribute 'hide'}
    bExecHome             : BOOL;
    {attribute 'hide'}
    bNewMoveReq           : BOOL;
    {attribute 'hide'}
    bHomeBusy             : BOOL;
    {attribute 'hide'}
    bPrepareDisable       : BOOL;
    {attribute 'hide'}
    bStepMoveDone         : BOOL;
    {attribute 'hide'}
    bStepMoveBusy         : BOOL;
    {attribute 'hide'}
    bHalt                 : BOOL;
    {attribute 'hide'}
    bOperational          : BOOL;
    {attribute 'hide'}
    bLimOverride          : BOOL;
    {attribute 'hide'}
    bPositionHold         : BOOL;
    {attribute 'hide'}
    bLocalExec            : BOOL;
    {attribute 'hide'}
    bSystemInit           : BOOL;
    {attribute 'hide'}
    bHomeDone             : BOOL;
    {attribute 'hide'}
    bCalibrationModeEnabled : BOOL;
    {attribute 'hide'}
    bStepModeEnabled         : BOOL;
    {attribute 'hide'}
    bHomeModeEnabled         : BOOL;
    {attribute 'hide'}
    bCSPModeEnabled          : BOOL;
    {attribute 'hide'}
    bSteModeEnable           : BOOL;
    {attribute 'hide'}
    bRestoreLoad             : BOOL;
    {attribute 'hide'}
    bStepModeParamsSet   : BOOL;
    {attribute 'hide'}
    bCalibrationAborted : BOOL;
    {attribute 'hide'}
    bCalibrationDone : BOOL;
    {attribute 'hide'}
    bExecParamsRead          : BOOL;
    {attribute 'hide'}
    bCommandMoveAbsolute     : BOOL;
    {attribute 'hide'}
    bRecentEnPosLagStatus    : BOOL;
    {attribute 'hide'}
    bDS402ManualAborted      : BOOL;
    {attribute 'hide'}
    bStepMoveAborted         : BOOL;
    {attribute 'hide'}
    bHomeAborted             : BOOL;
    {attribute 'hide'}
    bDS402Manual      : BOOL;
    {attribute 'hide'}
    bReset              : BOOL;
    {attribute 'hide'}
    nCmdDataLocal            : INT;
    {attribute 'hide'}
    bManualTransition        : BOOL;
    // ====== Measurements & scaled values ======
    {attribute 'hide'}
    nScaledFErrWin      : DINT;
    {attribute 'hide'}
    nScalededSteps      : DINT;
    {attribute 'hide'}
    fScalededSteps           : LREAL;
    {attribute 'hide'}
    fMeasuredVelo            : LREAL;
    {attribute 'hide'}
    fMeasuredAcc             : LREAL;
    {attribute 'hide'}
    fParameterValue          : LREAL;
    {attribute 'hide'}
    fMeasuredPos             : LREAL;
    // ====== Internal numeric parameters ======
    {attribute 'hide'}
    nScalededStepAmp         : UINT;
    {attribute 'hide'}
    nScaledStepFreq          : UINT;
    // ====== Timer and trigger FBs ======
    {attribute 'hide'}
    tonInitTimer             : TON;
    {attribute 'hide'}
    tonSyncHoming            : TON;
    {attribute 'hide'}
    tonHoldTime              : TON;
    {attribute 'hide'}
    tonSlowParamReadTimer    : TON;
    {attribute 'hide'}
    NCParamsTimer            : TON;
    {attribute 'hide'}
    tonRestoreRetry          : TON;

    {attribute 'hide'}
    rtExec                   : R_TRIG;
    {attribute 'hide'}
    rtMoveCmdShortcut        : R_TRIG;
    {attribute 'hide'}
    rtHomeCmdShortcut        : R_TRIG;
    {attribute 'hide'}
    rtEnableMode             : R_TRIG;
    {attribute 'hide'}
    rtUserExec               : R_TRIG;
    {attribute 'hide'}
    rtModeChange             : R_TRIG;
    {attribute 'hide'}
    rtMoveDone               : R_TRIG;
    {attribute 'hide'}
    rtNewMoveReq             : R_TRIG;
    {attribute 'hide'}
    ftExec                   : F_TRIG;
    {attribute 'hide'}
    rtCSPModeOk              : R_TRIG;
    {attribute 'hide'}
    rtHomeModeEnable         : R_TRIG;
    {attribute 'hide'}
    rtStepModeEnabled        : R_TRIG;
    {attribute 'hide'}
    rtNewServoMove           : R_TRIG;
    {attribute 'hide'}
    rtStepMove               : R_TRIG;
    rtHaltEdge : R_TRIG; // Rising edge for bHalt
    {attribute 'hide'}
    eDoneCause : E_MoveDoneCause := E_MoveDoneCause.Unknown;
    // ====== Channel-specific object indices ======
    nSubIndex                : BYTE := 0;        // Main subindex (which channel)
    {attribute 'hide'}
    nChanFErrWinIdx          : WORD;
    {attribute 'hide'}
    nChanSoftwareLimIdx      : WORD;
    {attribute 'hide'}
    nChanMotorLoadIdx        : WORD;
    {attribute 'hide'}
    nChanErrorCodeIdx        : WORD;
    {attribute 'hide'}
    nChanStepIdx             : WORD;
    {attribute 'hide'}
    nChanStepFreqIdx         : WORD;
    {attribute 'hide'}
    nChanStepAmpIdx          : WORD;
    {attribute 'hide'}
    nChanSoftLimitIdx        : WORD;
    {attribute 'hide'}
    nChanHomeOffsIdx         : WORD;
    {attribute 'hide'}
    nChanHomeVeloIdx         : WORD;
    {attribute 'hide'}
    nChanhomeAccIdx          : WORD;
    {attribute 'hide'}
    nMaxCloseLoopFreqIdx     : WORD;
    {attribute 'hide'}
    nPositionerTypeIdx       : WORD;
    {attribute 'hide'}
    nCalibrationOptIdx       : WORD;
    {attribute 'hide'}
    nSensorPowerModeIdx      : WORD;
    {attribute 'hide'}
    nReferencingOptIdx       : WORD;
    {attribute 'hide'}
    nReferenceTypeIdx        : WORD;
    {attribute 'hide'}
    nSafeDirIdx              : WORD;
    {attribute 'hide'}
    nMotorLoadIdx            : WORD;
    {attribute 'hide'}
    nChannelTypeIdx          : WORD;
    {attribute 'hide'}
    nChannelStateIdx         : WORD;
    {attribute 'hide'}
    nLogicalScaleOffsetIdx   : WORD;
    {attribute 'hide'}
    nLogicalScaleInvIdx      : WORD;
    {attribute 'hide'}
    rtStepCmdShortcut: R_TRIG;
    {attribute 'hide'}
    rtCalibrateCmdShortcut: R_TRIG;
    {attribute 'hide'}
    bCommandMoveStep: BOOL;
    {attribute 'hide'}
    bCalibrationsParamsSet: BOOL := TRUE;
    {attribute 'hide'}
    bHomingParamsSet: BOOL;
    {attribute 'hide'}
    bCalibrateMoveAborted: BOOL;
    {attribute 'hide'}
    bCalibrateMoveDone: BOOL;
    {attribute 'hide'}
    bChanParamsSet: BOOL;
    {attribute 'hide'}
    bCalibrationBusy: BOOL;
END_VAR

VAR CONSTANT
    {attribute 'hide'}
    nChanSoftLimitBase       : WORD := 16#200E;
    {attribute 'hide'}
    nHomeOffsetBase          : WORD := 16#607C;
    {attribute 'hide'}
    nHomingSpeedBase         : WORD := 16#6099;
    {attribute 'hide'}
    nhomingAccBase           : WORD := 16#609A;
    {attribute 'hide'}
    nErrorCodeBase           : WORD := 16#603F;
    {attribute 'hide'}
    nFErrWinBase             : WORD := 16#6065;
    {attribute 'hide'}
    nChanOfsBase             : WORD := 16#800;      // For SmartAct MCS2 and E-727
    {attribute 'hide'}
    nEncErrorCode            : WORD := 16#7300;     // Motor encoder defective code (for save/restore)
    {attribute 'hide'}
    nSoftLimBase             : WORD := 16#200E;
    {attribute 'hide'}
    nOlStepBase              : WORD := 16#2022;
    {attribute 'hide'}
    nOlStepAmpBase           : WORD := 16#2023;
    {attribute 'hide'}
    nOlStepFreqBase          : WORD := 16#2024;
    {attribute 'hide'}
    nMaxCloseLoopFreqBase    : WORD := 16#2001;
    {attribute 'hide'}
    nPositionerTypeBase      : WORD := 16#2000;
    {attribute 'hide'}
    nCalibrationOptBase      : WORD := 16#2004;
    {attribute 'hide'}
    nSensorPowerModeBase     : WORD := 16#2007;
    {attribute 'hide'}
    nReferencingOptBase      : WORD := 16#200B;
    {attribute 'hide'}
    nReferenceTypeBase       : WORD := 16#200A;
    {attribute 'hide'}
    nSafeDirBase             : WORD := 16#200C;
    {attribute 'hide'}
    nMotorLoadBase           : WORD := 16#200D;
    {attribute 'hide'}
    nChannelTypeBase         : WORD := 16#200F;
    {attribute 'hide'}
    nChannelStateBase        : WORD := 16#2025;
    {attribute 'hide'}
    nLogicalScaleOffsetBase  : WORD := 16#2008;
    {attribute 'hide'}
    nLogicalScaleInvBase     : WORD := 16#2009;
END_VAR

VAR PERSISTENT
    nCommandLocal            : INT;
    bSaved                   : BOOL;
    fSavedPosition           : LREAL;
END_VAR

IF NOT __ISVALIDREF( stMotionStage) THEN
    RETURN;
END_IF

// when the plc autoboot it appears reading from i/o is not yet after 'call_after_init'
IF bSystemInit THEN
    IF  stMotionStage.Axis.NcToPlc.AxisId <> 0 THEN
        stDS402Drive.nDS402DriveControl := 128; // clear errors, prepare for startup
        bExecParamsRead := TRUE; // trigger NC param read on first scan
        bSystemInit := FALSE;
    END_IF
END_IF
(* Check for the plc shortcut commands
   Used for testing or to circumvent motor record issues*)
rtMoveCmdShortcut(CLK:= stMotionStage.bMoveCmd);
rtHomeCmdShortcut(CLK:= stMotionStage.bHomeCmd);
rtStepCmdShortcut(CLK:= stMotionStage.stMCS2ChanParams.bStepMoveCmd);
rtCalibrateCmdShortcut(CLK:= stMotionStage.stMCS2ChanParams.bCalibrationCmd);

(* Execute on rising edge*)
IF rtMoveCmdShortcut.Q AND NOT stMotionStage.bExecute THEN
    stMotionStage.bExecute := TRUE;
    stMotionStage.nCommand := E_EpicsMotorCmd.MOVE_ABSOLUTE;
    bEnPosLag := bRecentEnPosLagStatus;
    fParameterValue := BOOL_TO_LREAL(bRecentEnPosLagStatus);

ELSIF rtStepCmdShortcut.Q AND NOT stMotionStage.bExecute THEN
    stMotionStage.bExecute := TRUE;
    stMotionStage.nCommand := E_EpicsMotorCmd.JOG;           // Step mode uses JOG
    nCommandLocal := E_EpicsMotorCmd.JOG;
    bEnPosLag := bRecentEnPosLagStatus;
    fParameterValue := BOOL_TO_LREAL(bRecentEnPosLagStatus);

ELSIF rtCalibrateCmdShortcut.Q AND NOT stMotionStage.bExecute THEN
    stMotionStage.bExecute := TRUE;
    stMotionStage.nCommand := E_EpicsMotorCmd.CALIBRATE;     // Calibration mode uses CALIBRATE
    nCommandLocal := E_EpicsMotorCmd.CALIBRATE;
    bEnPosLag := bRecentEnPosLagStatus;
    fParameterValue := BOOL_TO_LREAL(bRecentEnPosLagStatus);

ELSIF rtHomeCmdShortcut.Q AND NOT stMotionStage.bExecute THEN
    stMotionStage.bExecute := NOT (stMotionStage.nCmdData = E_EpicsHomeCmd.ABSOLUTE_SET)
                             OR NOT (stMotionStage.nCmdData = E_EpicsHomeCmd.NONE);
    stMotionStage.nCommand := E_EpicsMotorCmd.HOME;
    stMotionStage.nCmdData := stMotionStage.nHomingMode;
    IF stMotionStage.stAxisParameters.bCtrlEnablePosDiffControl.0 THEN
        bRecentEnPosLagStatus := stMotionStage.stAxisParameters.bCtrlEnablePosDiffControl.0;
        bEnPosLag := TRUE;
        fParameterValue := 0;
    END_IF
END_IF

(* entry point for local and EPICS main execs *)
rtUserExec(CLK:= stMotionStage.bExecute);
(* if a Move/Home Goal is comfirmed and there is no persistant
   error conditions, then we have a valid move request.*)
bNewMoveReq S= NOT  stMotionStage.bBusy AND rtUserExec.Q AND NOT  stMotionStage.bError;
(* this Move request is valid till an error occurs or the currently move is done *)
bNewMoveReq R= NOT  stMotionStage.bExecute OR  stMotionStage.bError;
bPrepareDisable R= bNewMoveReq;
rtNewMoveReq(CLK:=bNewMoveReq);
(* Moves are automatically allowed if no safety hooks.
   Otherwise, some other code will set this.*)
 stMotionStage.bSafetyReady :=  stMotionStage.bPowerSelf;
(* Set the proper command for the request move;
   if bservo not set, manual step moves will be performed *)
IF rtUserExec.Q THEN
    //  if we enter here form state movers
    stMotionStage.bMoveCmd := TRUE;
    nCommandLocal := E_EpicsMotorCmd.MOVE_ABSOLUTE;
    IF stMotionStage.bHomeCmd THEN
        nCommandLocal := stMotionStage.nCommand;
        nCmdDataLocal := stMotionStage.nCmdData;
    ELSIF stMotionStage.stMCS2ChanParams.bStepMoveCmd THEN
        // For stepmode, directly write the command
        stMotionStage.nCommand := E_EpicsMotorCmd.JOG;
        nCommandLocal := E_EpicsMotorCmd.JOG;
    ELSIF stMotionStage.stMCS2ChanParams.bCalibrationCmd THEN
        // For calibration, directly write the command
        stMotionStage.nCommand := E_EpicsMotorCmd.CALIBRATE;
        nCommandLocal := E_EpicsMotorCmd.CALIBRATE;
    END_IF

    IF NOT stMotionStage.bHomeCmd AND NOT stMotionStage.stMCS2ChanParams.stChannelState.bIsReferenced THEN
        // attempting to move an axis without homing first?
        IF stMotionStage.nHomingMode <> E_EpicsHomeCmd.NONE AND NOT stMotionStage.bHomed THEN
            stMotionStage.sErrorMessage := 'Axis homing mode set, but homing routine pending';
        END_IF
    END_IF
END_IF

(* Set the drive in the correct operating mode. based on requested move command!
    NB: bservo must set for close loop motion
*)
ModeOperation();

(* NB: This is the only tested mode of operation so far. also aligned
    piezo drive position holding feature
*)
rtEnableMode(CLK:=( stMotionStage.nEnableMode = E_StageEnableMode.DURING_MOTION));
(* Handle auto-enable timing *)
CASE  stMotionStage.nEnableMode OF
    (* Not recommended, not tested *)
    E_StageEnableMode.ALWAYS:
         stMotionStage.bEnable:=stMotionStage.bSafetyReady;
    E_StageEnableMode.DURING_MOTION:
        IF rtEnableMode.Q THEN
             stMotionStage.bEnable := FALSE;
        END_IF
        IF rtNewMoveReq.Q THEN
            (* override ongoing holding.*)
            bPositionHold := FALSE;
            tonHoldTime.IN:=FALSE;
            (*MC block are not compatible with open loop Motion
                thus we wathc for correct close loop modes to use NC features *)
             stMotionStage.bEnable :=  stMotionStage.bSafetyReady;
            bLastHoltTimeOut := FALSE;
            bHalt:=FALSE;
        END_IF
END_CASE
(*  Interlock mainly react on internal limit conditions inthe ove direction.
    MCS2 drive will go into error state when an internal limit is hit *)
Interlock();

